LIN {X 0,Y 600.839,Z 923.03,A -85,B 0,C 180,E1 7871.021,E2 7871.021} C_VEL
LIN {X 0,Y 600.811,Z 923.03,A -85,B 0,C 180,E1 7876.847,E2 7876.847} C_VEL
LIN {X 0,Y 600.932,Z 923.03,A -85,B 0,C 180,E1 7882.881,E2 7882.881} C_VEL
LIN {X 0,Y 600.969,Z 923.03,A -85,B 0,C 180,E1 7888.765,E2 7888.765} C_VEL
LIN {X 0,Y 601.067,Z 923.03,A -85,B 0,C 180,E1 7893.096,E2 7893.096} C_VEL
LIN {X 0,Y 601.172,Z 923.03,A -85,B 0,C 180,E1 7898.46,E2 7898.46} C_VEL
LIN {X 0,Y 601.119,Z 923.03,A -85,B 0,C 180,E1 7903.949,E2 7903.949} C_VEL
LIN {X 0,Y 601.484,Z 923.03,A -85,B 0,C 180,E1 7909.873,E2 7909.873} C_VEL
LIN {X 0,Y 601.549,Z 923.323,A -85,B 0,C 180,E1 7914.806,E2 7914.806} C_VEL
LIN {X 0,Y 606.229,Z 948.816,A -85,B 0,C 180,E1 7915.27,E2 7915.27} C_VEL
LIN {X 0,Y 606.178,Z 983.388,A -85,B 0,C 180,E1 7915.848,E2 7915.848} C_VEL
LIN {X 0,Y 605.698,Z 1012.075,A -85,B 0,C 180,E1 7916.874,E2 7916.874} C_VEL
LIN {X 0,Y 605.013,Z 1037.452,A -85,B 0,C 180,E1 7918.391,E2 7918.391} C_VEL
LIN {X 0,Y 604.292,Z 1059.313,A -85,B 0,C 180,E1 7920.36,E2 7920.36} C_VEL
LIN {X 0,Y 603.588,Z 1076.615,A -85,B 0,C 180,E1 7922.692,E2 7922.692} C_VEL
LIN {X 0,Y 602.997,Z 1089.111,A -85,B 0,C 180,E1 7925.394,E2 7925.394} C_VEL
LIN {X 0,Y 602.737,Z 1095.415,A -85,B 0,C 180,E1 7928.184,E2 7928.184} C_VEL
LIN {X 0,Y 602.671,Z 1096.34,A -85,B 0,C 180,E1 7930.11,E2 7930.11} C_VEL
LIN {X 0,Y 602.762,Z 1093.764,A -85,B 0,C 180,E1 7932.471,E2 7932.471} C_VEL
LIN {X 0,Y 602.992,Z 1086.371,A -85,B 0,C 180,E1 7934.97,E2 7934.97} C_VEL
LIN {X 0,Y 603.48,Z 1072.244,A -85,B 0,C 180,E1 7937.641,E2 7937.641} C_VEL
LIN {X 0,Y 604.098,Z 1054.164,A -85,B 0,C 180,E1 7939.855,E2 7939.855} C_VEL
LIN {X 0,Y 604.743,Z 1031.678,A -85,B 0,C 180,E1 7941.725,E2 7941.725} C_VEL
LIN {X 0,Y 605.526,Z 1005.59,A -85,B 0,C 180,E1 7943.163,E2 7943.163} C_VEL
LIN {X 0,Y 605.926,Z 976.016,A -85,B 0,C 180,E1 7944.13,E2 7944.13} C_VEL
LIN {X 0,Y 605.053,Z 940.656,A -85,B 0,C 180,E1 7944.678,E2 7944.678} C_VEL
LIN {X 0,Y 601.353,Z 923.03,A -85,B 0,C 180,E1 7945.032,E2 7945.032} C_VEL
LIN {X 0,Y 600.945,Z 923.03,A -85,B 0,C 180,E1 7951.231,E2 7951.231} C_VEL
LIN {X 0,Y 600.916,Z 923.03,A -85,B 0,C 180,E1 7957.124,E2 7957.124} C_VEL
LIN {X 0,Y 600.782,Z 923.03,A -85,B 0,C 180,E1 7963.15,E2 7963.15} C_VEL
LIN {X 0,Y 600.894,Z 923.03,A -85,B 0,C 180,E1 7969.157,E2 7969.157} C_VEL
LIN {X 0,Y 600.916,Z 923.03,A -85,B 0,C 180,E1 7974.652,E2 7974.652} C_VEL
LIN {X 0,Y 600.987,Z 923.03,A -85,B 0,C 180,E1 7979.798,E2 7979.798} C_VEL
LIN {X 0,Y 601.241,Z 923.03,A -85,B 0,C 180,E1 7984.798,E2 7984.798} C_VEL
LIN {X 0,Y 601.281,Z 923.03,A -85,B 0,C 180,E1 7990.919,E2 7990.919} C_VEL
LIN {X 0,Y 601.286,Z 923.03,A -85,B 0,C 180,E1 7995.433,E2 7995.433} C_VEL
LIN {X 0,Y 601.464,Z 923.03,A -85,B 0,C 180,E1 7999.859,E2 7999.859} C_VEL
LIN {X 0,Y 601.588,Z 923.03,A -85,B 0,C 180,E1 8004.221,E2 8004.221} C_VEL
LIN {X 0,Y 601.735,Z 923.03,A -85,B 0,C 180,E1 8008.548,E2 8008.548} C_VEL
LIN {X 0,Y 601.66,Z 923.03,A -85,B 0,C 180,E1 8012.866,E2 8012.866} C_VEL
LIN {X 0,Y 601.578,Z 923.03,A -85,B 0,C 180,E1 8017.202,E2 8017.202} C_VEL
LIN {X 0,Y 601.437,Z 923.03,A -85,B 0,C 180,E1 8023.055,E2 8023.055} C_VEL
LIN {X 0,Y 601.353,Z 923.03,A -85,B 0,C 180,E1 8027.535,E2 8027.535} C_VEL
LIN {X 0,Y 601.192,Z 923.03,A -85,B 0,C 180,E1 8032.134,E2 8032.134} C_VEL
LIN {X 0,Y 601.149,Z 923.03,A -85,B 0,C 180,E1 8036.885,E2 8036.885} C_VEL
LIN {X 0,Y 601.092,Z 923.03,A -85,B 0,C 180,E1 8041.847,E2 8041.847} C_VEL
LIN {X 0,Y 600.927,Z 923.03,A -85,B 0,C 180,E1 8047.101,E2 8047.101} C_VEL
LIN {X 0,Y 600.986,Z 923.03,A -85,B 0,C 180,E1 8053.181,E2 8053.181} C_VEL
LIN {X 0,Y 600.904,Z 923.03,A -85,B 0,C 180,E1 8059.167,E2 8059.167} C_VEL
LIN {X 0,Y 600.891,Z 923.03,A -85,B 0,C 180,E1 8064.66,E2 8064.66} C_VEL
LIN {X 0,Y 601.13,Z 923.03,A -85,B 0,C 180,E1 8070.645,E2 8070.645} C_VEL
LIN {X 0,Y 601.189,Z 923.03,A -85,B 0,C 180,E1 8071.123,E2 8071.123} C_VEL
LIN {X 0,Y 615.049,Z 964.555,A -85,B 0,C 180,E1 8072.72,E2 8072.72} C_VEL
LIN {X 0,Y 613.064,Z 1002.893,A -85,B 0,C 180,E1 8074.095,E2 8074.095} C_VEL
LIN {X 0,Y 610.732,Z 1039.044,A -85,B 0,C 180,E1 8075.978,E2 8075.978} C_VEL
LIN {X 0,Y 608.192,Z 1072.401,A -85,B 0,C 180,E1 8078.343,E2 8078.343} C_VEL
LIN {X 0,Y 605.791,Z 1103.466,A -85,B 0,C 180,E1 8081.305,E2 8081.305} C_VEL
LIN {X 0,Y 604.138,Z 1128.033,A -85,B 0,C 180,E1 8084.447,E2 8084.447} C_VEL
LIN {X 0,Y 602.911,Z 1147.172,A -85,B 0,C 180,E1 8087.731,E2 8087.731} C_VEL
LIN {X 0,Y 602.274,Z 1162.011,A -85,B 0,C 180,E1 8091.34,E2 8091.34} C_VEL
LIN {X 0,Y 601.991,Z 1171.367,A -85,B 0,C 180,E1 8094.958,E2 8094.958} C_VEL
LIN {X 0,Y 601.888,Z 1175.651,A -85,B 0,C 180,E1 8098.56,E2 8098.56} C_VEL
LIN {X 0,Y 601.892,Z 1175.605,A -85,B 0,C 180,E1 8101.437,E2 8101.437} C_VEL
LIN {X 0,Y 602.053,Z 1171.28,A -85,B 0,C 180,E1 8105.038,E2 8105.038} C_VEL
LIN {X 0,Y 602.289,Z 1161.868,A -85,B 0,C 180,E1 8108.656,E2 8108.656} C_VEL
LIN {X 0,Y 602.951,Z 1146.84,A -85,B 0,C 180,E1 8112.287,E2 8112.287} C_VEL
LIN {X 0,Y 604.213,Z 1126.109,A -85,B 0,C 180,E1 8115.767,E2 8115.767} C_VEL
LIN {X 0,Y 605.984,Z 1100.522,A -85,B 0,C 180,E1 8118.914,E2 8118.914} C_VEL
LIN {X 0,Y 608.17,Z 1070.791,A -85,B 0,C 180,E1 8121.65,E2 8121.65} C_VEL
LIN {X 0,Y 610.558,Z 1037.737,A -85,B 0,C 180,E1 8123.925,E2 8123.925} C_VEL
LIN {X 0,Y 612.697,Z 1001.543,A -85,B 0,C 180,E1 8125.747,E2 8125.747} C_VEL
LIN {X 0,Y 613.951,Z 963.531,A -85,B 0,C 180,E1 8127.081,E2 8127.081} C_VEL
LIN {X 0,Y 601.155,Z 923.03,A -85,B 0,C 180,E1 8128.626,E2 8128.626} C_VEL
LIN {X 0,Y 601.011,Z 923.03,A -85,B 0,C 180,E1 8133.962,E2 8133.962} C_VEL
LIN {X 0,Y 600.872,Z 923.03,A -85,B 0,C 180,E1 8138.953,E2 8138.953} C_VEL
LIN {X 0,Y 600.837,Z 923.03,A -85,B 0,C 180,E1 8140.89,E2 8140.89} C_VEL
LIN {X 0,Y 599.556,Z 923.03,A -85,B 0,C 180,E1 8141.715,E2 8141.715} C_VEL
LIN {X 0,Y 592.929,Z 923.03,A -85,B 0,C 180,E1 8143.956,E2 8143.956} C_VEL
LIN {X 0,Y 592.846,Z 923.03,A -85,B 0,C 180,E1 8144.169,E2 8144.169} C_VEL
LIN {X 0,Y 592.915,Z 923.03,A -85,B 0,C 180,E1 8149.867,E2 8149.867} C_VEL
LIN {X 0,Y 593.127,Z 923.03,A -85,B 0,C 180,E1 8154.61,E2 8154.61} C_VEL
LIN {X 0,Y 593.112,Z 923.03,A -85,B 0,C 180,E1 8160.269,E2 8160.269} C_VEL
LIN {X 0,Y 608.042,Z 967.522,A -85,B 0,C 180,E1 8161.664,E2 8161.664} C_VEL
LIN {X 0,Y 606.659,Z 1011.398,A -85,B 0,C 180,E1 8162.505,E2 8162.505} C_VEL
LIN {X 0,Y 604.629,Z 1052.765,A -85,B 0,C 180,E1 8163.898,E2 8163.898} C_VEL
LIN {X 0,Y 602.308,Z 1090.442,A -85,B 0,C 180,E1 8165.76,E2 8165.76} C_VEL
LIN {X 0,Y 599.934,Z 1125.316,A -85,B 0,C 180,E1 8168.121,E2 8168.121} C_VEL
LIN {X 0,Y 597.69,Z 1156.933,A -85,B 0,C 180,E1 8170.983,E2 8170.983} C_VEL
LIN {X 0,Y 595.986,Z 1183.561,A -85,B 0,C 180,E1 8174.209,E2 8174.209} C_VEL
LIN {X 0,Y 594.902,Z 1204.715,A -85,B 0,C 180,E1 8177.707,E2 8177.707} C_VEL
LIN {X 0,Y 594.348,Z 1219.788,A -85,B 0,C 180,E1 8181.239,E2 8181.239} C_VEL
LIN {X 0,Y 594.132,Z 1229.686,A -85,B 0,C 180,E1 8184.906,E2 8184.906} C_VEL
LIN {X 0,Y 594.006,Z 1234.224,A -85,B 0,C 180,E1 8188.555,E2 8188.555} C_VEL
LIN {X 0,Y 594.127,Z 1234.236,A -85,B 0,C 180,E1 8191.47,E2 8191.47} C_VEL
LIN {X 0,Y 594.141,Z 1229.748,A -85,B 0,C 180,E1 8195.119,E2 8195.119} C_VEL
LIN {X 0,Y 594.374,Z 1219.948,A -85,B 0,C 180,E1 8198.786,E2 8198.786} C_VEL
LIN {X 0,Y 594.984,Z 1204.01,A -85,B 0,C 180,E1 8202.536,E2 8202.536} C_VEL
LIN {X 0,Y 596.173,Z 1183.005,A -85,B 0,C 180,E1 8206.006,E2 8206.006} C_VEL
LIN {X 0,Y 597.992,Z 1157.056,A -85,B 0,C 180,E1 8209.19,E2 8209.19} C_VEL
LIN {X 0,Y 600.341,Z 1126.206,A -85,B 0,C 180,E1 8212.046,E2 8212.046} C_VEL
LIN {X 0,Y 602.999,Z 1091.774,A -85,B 0,C 180,E1 8214.435,E2 8214.435} C_VEL
LIN {X 0,Y 605.496,Z 1055.147,A -85,B 0,C 180,E1 8216.294,E2 8216.294} C_VEL
LIN {X 0,Y 607.732,Z 1015.786,A -85,B 0,C 180,E1 8217.658,E2 8217.658} C_VEL
LIN {X 0,Y 609.171,Z 974.132,A -85,B 0,C 180,E1 8218.5,E2 8218.5} C_VEL
LIN {X 0,Y 608.398,Z 964.807,A -85,B 0,C 180,E1 8218.666,E2 8218.666} C_VEL
LIN {X 0,Y 593.159,Z 923.03,A -85,B 0,C 180,E1 8219.987,E2 8219.987} C_VEL
LIN {X 0,Y 593.061,Z 923.03,A -85,B 0,C 180,E1 8225.888,E2 8225.888} C_VEL
LIN {X 0,Y 592.896,Z 923.03,A -85,B 0,C 180,E1 8231.515,E2 8231.515} C_VEL
LIN {X 0,Y 592.87,Z 923.03,A -85,B 0,C 180,E1 8236.517,E2 8236.517} C_VEL
LIN {X 0,Y 592.972,Z 923.03,A -85,B 0,C 180,E1 8242.297,E2 8242.297} C_VEL
LIN {X 0,Y 593.014,Z 923.03,A -85,B 0,C 180,E1 8247.65,E2 8247.65} C_VEL
LIN {X 0,Y 593.197,Z 923.03,A -85,B 0,C 180,E1 8253.09,E2 8253.09} C_VEL
LIN {X 0,Y 593.241,Z 923.03,A -85,B 0,C 180,E1 8257.539,E2 8257.539} C_VEL
LIN {X 0,Y 593.162,Z 923.03,A -85,B 0,C 180,E1 8262.201,E2 8262.201} C_VEL
LIN {X 0,Y 593.359,Z 923.03,A -85,B 0,C 180,E1 8266.752,E2 8266.752} C_VEL
LIN {X 0,Y 593.633,Z 923.03,A -85,B 0,C 180,E1 8271.216,E2 8271.216} C_VEL
LIN {X 0,Y 593.674,Z 923.03,A -85,B 0,C 180,E1 8274.57,E2 8274.57} C_VEL
LIN {X 0,Y 598.641,Z 949.1,A -85,B 0,C 180,E1 8275.069,E2 8275.069} C_VEL
LIN {X 0,Y 598.556,Z 985.6,A -85,B 0,C 180,E1 8275.704,E2 8275.704} C_VEL
LIN {X 0,Y 597.994,Z 1014.937,A -85,B 0,C 180,E1 8276.799,E2 8276.799} C_VEL
LIN {X 0,Y 597.269,Z 1040.755,A -85,B 0,C 180,E1 8278.416,E2 8278.416} C_VEL
LIN {X 0,Y 596.536,Z 1061.495,A -85,B 0,C 180,E1 8280.364,E2 8280.364} C_VEL
LIN {X 0,Y 595.798,Z 1078.379,A -85,B 0,C 180,E1 8282.727,E2 8282.727} C_VEL
LIN {X 0,Y 595.178,Z 1090.542,A -85,B 0,C 180,E1 8285.465,E2 8285.465} C_VEL
LIN {X 0,Y 594.942,Z 1095.937,A -85,B 0,C 180,E1 8287.823,E2 8287.823} C_VEL
LIN {X 0,Y 594.827,Z 1097.225,A -85,B 0,C 180,E1 8290.245,E2 8290.245} C_VEL
LIN {X 0,Y 594.927,Z 1094.162,A -85,B 0,C 180,E1 8292.718,E2 8292.718} C_VEL
LIN {X 0,Y 595.185,Z 1086.391,A -85,B 0,C 180,E1 8295.225,E2 8295.225} C_VEL
LIN {X 0,Y 595.693,Z 1073.073,A -85,B 0,C 180,E1 8297.724,E2 8297.724} C_VEL
LIN {X 0,Y 596.316,Z 1055.103,A -85,B 0,C 180,E1 8299.948,E2 8299.948} C_VEL
LIN {X 0,Y 597,Z 1032.853,A -85,B 0,C 180,E1 8301.826,E2 8301.826} C_VEL
LIN {X 0,Y 597.811,Z 1006.241,A -85,B 0,C 180,E1 8303.312,E2 8303.312} C_VEL
LIN {X 0,Y 598.239,Z 977.995,A -85,B 0,C 180,E1 8304.258,E2 8304.258} C_VEL
LIN {X 0,Y 597.427,Z 942.053,A -85,B 0,C 180,E1 8304.83,E2 8304.83} C_VEL
LIN {X 0,Y 593.406,Z 923.03,A -85,B 0,C 180,E1 8305.245,E2 8305.245} C_VEL
LIN {X 0,Y 593.037,Z 923.03,A -85,B 0,C 180,E1 8310.64,E2 8310.64} C_VEL
LIN {X 0,Y 593.023,Z 923.03,A -85,B 0,C 180,E1 8315.88,E2 8315.88} C_VEL
LIN {X 0,Y 592.86,Z 923.03,A -85,B 0,C 180,E1 8321.508,E2 8321.508} C_VEL
LIN {X 0,Y 592.881,Z 923.03,A -85,B 0,C 180,E1 8326.503,E2 8326.503} C_VEL
LIN {X 0,Y 592.974,Z 923.03,A -85,B 0,C 180,E1 8332.283,E2 8332.283} C_VEL
LIN {X 0,Y 593,Z 923.03,A -85,B 0,C 180,E1 8337.636,E2 8337.636} C_VEL
LIN {X 0,Y 593.274,Z 923.03,A -85,B 0,C 180,E1 8343.062,E2 8343.062} C_VEL
LIN {X 0,Y 593.316,Z 923.03,A -85,B 0,C 180,E1 8349.099,E2 8349.099} C_VEL
LIN {X 0,Y 593.421,Z 923.03,A -85,B 0,C 180,E1 8353.722,E2 8353.722} C_VEL
LIN {X 0,Y 593.567,Z 923.03,A -85,B 0,C 180,E1 8359.723,E2 8359.723} C_VEL
LIN {X 0,Y 593.68,Z 923.03,A -85,B 0,C 180,E1 8364.144,E2 8364.144} C_VEL
LIN {X 0,Y 593.835,Z 923.03,A -85,B 0,C 180,E1 8368.529,E2 8368.529} C_VEL
LIN {X 0,Y 593.757,Z 923.03,A -85,B 0,C 180,E1 8372.904,E2 8372.904} C_VEL
LIN {X 0,Y 593.69,Z 923.03,A -85,B 0,C 180,E1 8377.298,E2 8377.298} C_VEL
LIN {X 0,Y 593.515,Z 923.03,A -85,B 0,C 180,E1 8383.232,E2 8383.232} C_VEL
LIN {X 0,Y 593.417,Z 923.03,A -85,B 0,C 180,E1 8387.777,E2 8387.777} C_VEL
LIN {X 0,Y 593.266,Z 923.03,A -85,B 0,C 180,E1 8393.512,E2 8393.512} C_VEL
LIN {X 0,Y 593.163,Z 923.03,A -85,B 0,C 180,E1 8398.931,E2 8398.931} C_VEL
LIN {X 0,Y 593.076,Z 923.03,A -85,B 0,C 180,E1 8404.074,E2 8404.074} C_VEL
LIN {X 0,Y 592.976,Z 923.03,A -85,B 0,C 180,E1 8410.135,E2 8410.135} C_VEL
LIN {X 0,Y 593.042,Z 923.03,A -85,B 0,C 180,E1 8415.493,E2 8415.493} C_VEL
LIN {X 0,Y 592.96,Z 923.03,A -85,B 0,C 180,E1 8420.422,E2 8420.422} C_VEL
LIN {X 0,Y 592.984,Z 923.03,A -85,B 0,C 180,E1 8425.899,E2 8425.899} C_VEL
LIN {X 0,Y 593.252,Z 923.03,A -85,B 0,C 180,E1 8430.77,E2 8430.77} C_VEL
LIN {X 0,Y 606.588,Z 962.66,A -85,B 0,C 180,E1 8432.292,E2 8432.292} C_VEL
LIN {X 0,Y 607.639,Z 971.467,A -85,B 0,C 180,E1 8432.613,E2 8432.613} C_VEL
LIN {X 0,Y 605.368,Z 1010.118,A -85,B 0,C 180,E1 8434.12,E2 8434.12} C_VEL
LIN {X 0,Y 602.904,Z 1045.237,A -85,B 0,C 180,E1 8436.081,E2 8436.081} C_VEL
LIN {X 0,Y 600.27,Z 1077.861,A -85,B 0,C 180,E1 8438.542,E2 8438.542} C_VEL
LIN {X 0,Y 597.891,Z 1106.529,A -85,B 0,C 180,E1 8441.413,E2 8441.413} C_VEL
LIN {X 0,Y 596.236,Z 1130.448,A -85,B 0,C 180,E1 8444.595,E2 8444.595} C_VEL
LIN {X 0,Y 595.021,Z 1149.05,A -85,B 0,C 180,E1 8447.921,E2 8447.921} C_VEL
LIN {X 0,Y 594.384,Z 1163.562,A -85,B 0,C 180,E1 8451.63,E2 8451.63} C_VEL
LIN {X 0,Y 594.104,Z 1171.715,A -85,B 0,C 180,E1 8454.891,E2 8454.891} C_VEL
LIN {X 0,Y 593.997,Z 1176.028,A -85,B 0,C 180,E1 8458.541,E2 8458.541} C_VEL
LIN {X 0,Y 594.002,Z 1175.994,A -85,B 0,C 180,E1 8461.456,E2 8461.456} C_VEL
LIN {X 0,Y 594.166,Z 1171.662,A -85,B 0,C 180,E1 8465.105,E2 8465.105} C_VEL
LIN {X 0,Y 594.432,Z 1162.222,A -85,B 0,C 180,E1 8468.772,E2 8468.772} C_VEL
LIN {X 0,Y 595.182,Z 1147.096,A -85,B 0,C 180,E1 8472.45,E2 8472.45} C_VEL
LIN {X 0,Y 596.513,Z 1125.857,A -85,B 0,C 180,E1 8476.029,E2 8476.029} C_VEL
LIN {X 0,Y 598.377,Z 1100.484,A -85,B 0,C 180,E1 8479.164,E2 8479.164} C_VEL
LIN {X 0,Y 600.701,Z 1070.721,A -85,B 0,C 180,E1 8481.922,E2 8481.922} C_VEL
LIN {X 0,Y 603.145,Z 1038.13,A -85,B 0,C 180,E1 8484.186,E2 8484.186} C_VEL
LIN {X 0,Y 605.376,Z 1002.436,A -85,B 0,C 180,E1 8486.008,E2 8486.008} C_VEL
LIN {X 0,Y 606.568,Z 965.188,A -85,B 0,C 180,E1 8487.351,E2 8487.351} C_VEL
LIN {X 0,Y 593.251,Z 923.03,A -85,B 0,C 180,E1 8489.01,E2 8489.01} C_VEL
LIN {X 0,Y 593.096,Z 923.03,A -85,B 0,C 180,E1 8494.09,E2 8494.09} C_VEL
LIN {X 0,Y 592.889,Z 923.03,A -85,B 0,C 180,E1 8500.154,E2 8500.154} C_VEL
LIN {X 0,Y 592.846,Z 923.03,A -85,B 0,C 180,E1 8504.169,E2 8504.169} C_VEL
LIN {X 0,Y 590.332,Z 923.03,A -85,B 0,C 180,E1 8505.418,E2 8505.418} C_VEL
LIN {X 0,Y 585.013,Z 923.03,A -85,B 0,C 180,E1 8507.288,E2 8507.288} C_VEL
LIN {X 0,Y 584.936,Z 923.03,A -85,B 0,C 180,E1 8507.504,E2 8507.504} C_VEL
LIN {X 0,Y 585.103,Z 923.03,A -85,B 0,C 180,E1 8513.579,E2 8513.579} C_VEL
LIN {X 0,Y 585.108,Z 923.03,A -85,B 0,C 180,E1 8518.919,E2 8518.919} C_VEL
LIN {X 0,Y 585.221,Z 923.832,A -85,B 0,C 180,E1 8519.878,E2 8519.878} C_VEL
LIN {X 0,Y 600.717,Z 968.424,A -85,B 0,C 180,E1 8521.349,E2 8521.349} C_VEL
LIN {X 0,Y 599.355,Z 1012.032,A -85,B 0,C 180,E1 8522.228,E2 8522.228} C_VEL
LIN {X 0,Y 597.227,Z 1051.908,A -85,B 0,C 180,E1 8523.592,E2 8523.592} C_VEL
LIN {X 0,Y 594.872,Z 1088.957,A -85,B 0,C 180,E1 8525.437,E2 8525.437} C_VEL
LIN {X 0,Y 592.385,Z 1123.725,A -85,B 0,C 180,E1 8527.799,E2 8527.799} C_VEL
LIN {X 0,Y 590.099,Z 1154.409,A -85,B 0,C 180,E1 8530.571,E2 8530.571} C_VEL
LIN {X 0,Y 588.384,Z 1179.9,A -85,B 0,C 180,E1 8533.605,E2 8533.605} C_VEL
LIN {X 0,Y 587.153,Z 1201.242,A -85,B 0,C 180,E1 8537.001,E2 8537.001} C_VEL
LIN {X 0,Y 586.533,Z 1216.535,A -85,B 0,C 180,E1 8540.374,E2 8540.374} C_VEL
LIN {X 0,Y 586.243,Z 1227.644,A -85,B 0,C 180,E1 8544.096,E2 8544.096} C_VEL
LIN {X 0,Y 586.156,Z 1232.583,A -85,B 0,C 180,E1 8547.058,E2 8547.058} C_VEL
LIN {X 0,Y 586.159,Z 1234.269,A -85,B 0,C 180,E1 8550.013,E2 8550.013} C_VEL
LIN {X 0,Y 586.142,Z 1231.745,A -85,B 0,C 180,E1 8553.708,E2 8553.708} C_VEL
LIN {X 0,Y 586.328,Z 1224.067,A -85,B 0,C 180,E1 8557.416,E2 8557.416} C_VEL
LIN {X 0,Y 586.802,Z 1210.807,A -85,B 0,C 180,E1 8561.148,E2 8561.148} C_VEL
LIN {X 0,Y 587.819,Z 1191.119,A -85,B 0,C 180,E1 8564.908,E2 8564.908} C_VEL
LIN {X 0,Y 589.562,Z 1165.631,A -85,B 0,C 180,E1 8568.406,E2 8568.406} C_VEL
LIN {X 0,Y 591.892,Z 1137.261,A -85,B 0,C 180,E1 8571.328,E2 8571.328} C_VEL
LIN {X 0,Y 594.48,Z 1104.527,A -85,B 0,C 180,E1 8573.883,E2 8573.883} C_VEL
LIN {X 0,Y 597.256,Z 1068.104,A -85,B 0,C 180,E1 8575.985,E2 8575.985} C_VEL
LIN {X 0,Y 599.829,Z 1029.624,A -85,B 0,C 180,E1 8577.542,E2 8577.542} C_VEL
LIN {X 0,Y 601.584,Z 990.606,A -85,B 0,C 180,E1 8578.549,E2 8578.549} C_VEL
LIN {X 0,Y 601.473,Z 967.455,A -85,B 0,C 180,E1 8578.945,E2 8578.945} C_VEL
LIN {X 0,Y 585.234,Z 923.03,A -85,B 0,C 180,E1 8580.427,E2 8580.427} C_VEL
LIN {X 0,Y 585.173,Z 923.03,A -85,B 0,C 180,E1 8584.631,E2 8584.631} C_VEL
LIN {X 0,Y 585.011,Z 923.03,A -85,B 0,C 180,E1 8590.235,E2 8590.235} C_VEL
LIN {X 0,Y 584.963,Z 923.03,A -85,B 0,C 180,E1 8596.341,E2 8596.341} C_VEL
LIN {X 0,Y 585.009,Z 923.03,A -85,B 0,C 180,E1 8601.691,E2 8601.691} C_VEL
LIN {X 0,Y 585.106,Z 923.03,A -85,B 0,C 180,E1 8607.158,E2 8607.158} C_VEL
LIN {X 0,Y 585.178,Z 923.03,A -85,B 0,C 180,E1 8612.304,E2 8612.304} C_VEL
LIN {X 0,Y 585.319,Z 923.03,A -85,B 0,C 180,E1 8617.218,E2 8617.218} C_VEL
LIN {X 0,Y 585.267,Z 923.03,A -85,B 0,C 180,E1 8622.831,E2 8622.831} C_VEL
LIN {X 0,Y 585.575,Z 923.03,A -85,B 0,C 180,E1 8628.736,E2 8628.736} C_VEL
LIN {X 0,Y 585.764,Z 923.03,A -85,B 0,C 180,E1 8634.311,E2 8634.311} C_VEL
LIN {X 0,Y 591.065,Z 950.012,A -85,B 0,C 180,E1 8634.868,E2 8634.868} C_VEL
LIN {X 0,Y 590.958,Z 986.526,A -85,B 0,C 180,E1 8635.51,E2 8635.51} C_VEL
LIN {X 0,Y 590.378,Z 1015.616,A -85,B 0,C 180,E1 8636.608,E2 8636.608} C_VEL
LIN {X 0,Y 589.616,Z 1041.655,A -85,B 0,C 180,E1 8638.258,E2 8638.258} C_VEL
LIN {X 0,Y 588.859,Z 1062.054,A -85,B 0,C 180,E1 8640.185,E2 8640.185} C_VEL
LIN {X 0,Y 588.043,Z 1079.108,A -85,B 0,C 180,E1 8642.579,E2 8642.579} C_VEL
LIN {X 0,Y 587.414,Z 1090.749,A -85,B 0,C 180,E1 8645.167,E2 8645.167} C_VEL
LIN {X 0,Y 587.143,Z 1096.322,A -85,B 0,C 180,E1 8647.395,E2 8647.395} C_VEL
LIN {X 0,Y 586.992,Z 1098.11,A -85,B 0,C 180,E1 8650.383,E2 8650.383} C_VEL
LIN {X 0,Y 587.1,Z 1094.473,A -85,B 0,C 180,E1 8652.979,E2 8652.979} C_VEL
LIN {X 0,Y 587.437,Z 1085.55,A -85,B 0,C 180,E1 8655.682,E2 8655.682} C_VEL
LIN {X 0,Y 588.003,Z 1070.16,A -85,B 0,C 180,E1 8658.35,E2 8658.35} C_VEL
LIN {X 0,Y 588.748,Z 1051.052,A -85,B 0,C 180,E1 8660.532,E2 8660.532} C_VEL
LIN {X 0,Y 589.522,Z 1026.602,A -85,B 0,C 180,E1 8662.415,E2 8662.415} C_VEL
LIN {X 0,Y 590.225,Z 998.779,A -85,B 0,C 180,E1 8663.797,E2 8663.797} C_VEL
LIN {X 0,Y 590.596,Z 967.955,A -85,B 0,C 180,E1 8664.628,E2 8664.628} C_VEL
LIN {X 0,Y 589.648,Z 942.756,A -85,B 0,C 180,E1 8664.996,E2 8664.996} C_VEL
LIN {X 0,Y 585.47,Z 923.03,A -85,B 0,C 180,E1 8665.379,E2 8665.379} C_VEL
LIN {X 0,Y 585.053,Z 923.03,A -85,B 0,C 180,E1 8671.517,E2 8671.517} C_VEL
LIN {X 0,Y 585.033,Z 923.03,A -85,B 0,C 180,E1 8676.788,E2 8676.788} C_VEL
LIN {X 0,Y 584.943,Z 923.03,A -85,B 0,C 180,E1 8682.198,E2 8682.198} C_VEL
LIN {X 0,Y 584.998,Z 923.03,A -85,B 0,C 180,E1 8687.797,E2 8687.797} C_VEL
LIN {X 0,Y 585.039,Z 923.03,A -85,B 0,C 180,E1 8693.542,E2 8693.542} C_VEL
LIN {X 0,Y 585.103,Z 923.03,A -85,B 0,C 180,E1 8698.889,E2 8698.889} C_VEL
LIN {X 0,Y 585.331,Z 923.03,A -85,B 0,C 180,E1 8704.634,E2 8704.634} C_VEL
LIN {X 0,Y 585.43,Z 923.03,A -85,B 0,C 180,E1 8710.382,E2 8710.382} C_VEL
LIN {X 0,Y 585.46,Z 923.03,A -85,B 0,C 180,E1 8715.03,E2 8715.03} C_VEL
LIN {X 0,Y 585.643,Z 923.03,A -85,B 0,C 180,E1 8719.582,E2 8719.582} C_VEL
LIN {X 0,Y 585.806,Z 923.03,A -85,B 0,C 180,E1 8724.065,E2 8724.065} C_VEL
LIN {X 0,Y 585.934,Z 923.03,A -85,B 0,C 180,E1 8728.509,E2 8728.509} C_VEL
LIN {X 0,Y 585.856,Z 923.03,A -85,B 0,C 180,E1 8732.944,E2 8732.944} C_VEL
LIN {X 0,Y 585.776,Z 923.03,A -85,B 0,C 180,E1 8737.397,E2 8737.397} C_VEL
LIN {X 0,Y 585.608,Z 923.03,A -85,B 0,C 180,E1 8743.414,E2 8743.414} C_VEL
LIN {X 0,Y 585.502,Z 923.03,A -85,B 0,C 180,E1 8748.026,E2 8748.026} C_VEL
LIN {X 0,Y 585.335,Z 923.03,A -85,B 0,C 180,E1 8752.766,E2 8752.766} C_VEL
LIN {X 0,Y 585.264,Z 923.03,A -85,B 0,C 180,E1 8758.613,E2 8758.613} C_VEL
LIN {X 0,Y 585.164,Z 923.03,A -85,B 0,C 180,E1 8764.599,E2 8764.599} C_VEL
LIN {X 0,Y 585.076,Z 923.03,A -85,B 0,C 180,E1 8770.195,E2 8770.195} C_VEL
LIN {X 0,Y 585.132,Z 923.03,A -85,B 0,C 180,E1 8775.789,E2 8775.789} C_VEL
LIN {X 0,Y 585.002,Z 923.03,A -85,B 0,C 180,E1 8781.687,E2 8781.687} C_VEL
LIN {X 0,Y 585.079,Z 923.03,A -85,B 0,C 180,E1 8787.153,E2 8787.153} C_VEL
LIN {X 0,Y 585.351,Z 923.785,A -85,B 0,C 180,E1 8790.407,E2 8790.407} C_VEL
LIN {X 0,Y 598.951,Z 963.422,A -85,B 0,C 180,E1 8791.971,E2 8791.971} C_VEL
LIN {X 0,Y 600.452,Z 971.844,A -85,B 0,C 180,E1 8792.307,E2 8792.307} C_VEL
LIN {X 0,Y 598.023,Z 1010.969,A -85,B 0,C 180,E1 8793.856,E2 8793.856} C_VEL
LIN {X 0,Y 595.384,Z 1046.785,A -85,B 0,C 180,E1 8795.894,E2 8795.894} C_VEL
LIN {X 0,Y 592.716,Z 1078.64,A -85,B 0,C 180,E1 8798.34,E2 8798.34} C_VEL
LIN {X 0,Y 590.187,Z 1107.402,A -85,B 0,C 180,E1 8801.266,E2 8801.266} C_VEL
LIN {X 0,Y 588.497,Z 1130.788,A -85,B 0,C 180,E1 8804.423,E2 8804.423} C_VEL
LIN {X 0,Y 587.176,Z 1149.703,A -85,B 0,C 180,E1 8807.853,E2 8807.853} C_VEL
LIN {X 0,Y 586.52,Z 1163.737,A -85,B 0,C 180,E1 8811.479,E2 8811.479} C_VEL
LIN {X 0,Y 586.219,Z 1172.062,A -85,B 0,C 180,E1 8814.822,E2 8814.822} C_VEL
LIN {X 0,Y 586.127,Z 1176.404,A -85,B 0,C 180,E1 8818.521,E2 8818.521} C_VEL
LIN {X 0,Y 586.132,Z 1176.382,A -85,B 0,C 180,E1 8821.476,E2 8821.476} C_VEL
LIN {X 0,Y 586.295,Z 1172.039,A -85,B 0,C 180,E1 8825.174,E2 8825.174} C_VEL
LIN {X 0,Y 586.587,Z 1162.566,A -85,B 0,C 180,E1 8828.89,E2 8828.89} C_VEL
LIN {X 0,Y 587.409,Z 1146.94,A -85,B 0,C 180,E1 8832.695,E2 8832.695} C_VEL
LIN {X 0,Y 588.832,Z 1125.985,A -85,B 0,C 180,E1 8836.244,E2 8836.244} C_VEL
LIN {X 0,Y 590.779,Z 1100.486,A -85,B 0,C 180,E1 8839.42,E2 8839.42} C_VEL
LIN {X 0,Y 593.185,Z 1071.329,A -85,B 0,C 180,E1 8842.151,E2 8842.151} C_VEL
LIN {X 0,Y 595.732,Z 1038.857,A -85,B 0,C 180,E1 8844.44,E2 8844.44} C_VEL
LIN {X 0,Y 598.151,Z 1002.052,A -85,B 0,C 180,E1 8846.338,E2 8846.338} C_VEL
LIN {X 0,Y 599.29,Z 967.203,A -85,B 0,C 180,E1 8847.619,E2 8847.619} C_VEL
LIN {X 0,Y 586.769,Z 927.616,A -85,B 0,C 180,E1 8849.206,E2 8849.206} C_VEL
LIN {X 0,Y 585.356,Z 923.03,A -85,B 0,C 180,E1 8849.371,E2 8849.371} C_VEL
LIN {X 0,Y 585.171,Z 923.03,A -85,B 0,C 180,E1 8854.617,E2 8854.617} C_VEL
LIN {X 0,Y 584.987,Z 923.03,A -85,B 0,C 180,E1 8860.222,E2 8860.222} C_VEL
LIN {X 0,Y 584.965,Z 923.03,A -85,B 0,C 180,E1 8866.326,E2 8866.326} C_VEL
LIN {X 0,Y 584.936,Z 923.03,A -85,B 0,C 180,E1 8867.504,E2 8867.504} C_VEL
LIN {X 0,Y 582.445,Z 923.03,A -85,B 0,C 180,E1 8868.768,E2 8868.768} C_VEL
LIN {X 0,Y 577.15,Z 923.03,A -85,B 0,C 180,E1 8870.66,E2 8870.66} C_VEL
LIN {X 0,Y 577.081,Z 923.03,A -85,B 0,C 180,E1 8870.879,E2 8870.879} C_VEL
LIN {X 0,Y 577.206,Z 923.03,A -85,B 0,C 180,E1 8876.9,E2 8876.9} C_VEL
LIN {X 0,Y 577.239,Z 923.115,A -85,B 0,C 180,E1 8879.405,E2 8879.405} C_VEL
LIN {X 0,Y 591.158,Z 963.17,A -85,B 0,C 180,E1 8880.816,E2 8880.816} C_VEL
LIN {X 0,Y 593.655,Z 973.013,A -85,B 0,C 180,E1 8881.095,E2 8881.095} C_VEL
LIN {X 0,Y 591.963,Z 1015.439,A -85,B 0,C 180,E1 8882.019,E2 8882.019} C_VEL
LIN {X 0,Y 589.617,Z 1056.219,A -85,B 0,C 180,E1 8883.499,E2 8883.499} C_VEL
LIN {X 0,Y 586.973,Z 1094.02,A -85,B 0,C 180,E1 8885.49,E2 8885.49} C_VEL
LIN {X 0,Y 584.262,Z 1129.871,A -85,B 0,C 180,E1 8888.091,E2 8888.091} C_VEL
LIN {X 0,Y 581.948,Z 1159.976,A -85,B 0,C 180,E1 8891.012,E2 8891.012} C_VEL
LIN {X 0,Y 580.241,Z 1184.592,A -85,B 0,C 180,E1 8894.165,E2 8894.165} C_VEL
LIN {X 0,Y 579.127,Z 1204.486,A -85,B 0,C 180,E1 8897.584,E2 8897.584} C_VEL
LIN {X 0,Y 578.557,Z 1219.966,A -85,B 0,C 180,E1 8901.377,E2 8901.377} C_VEL
LIN {X 0,Y 578.373,Z 1228.808,A -85,B 0,C 180,E1 8904.767,E2 8904.767} C_VEL
LIN {X 0,Y 578.234,Z 1233.434,A -85,B 0,C 180,E1 8908.516,E2 8908.516} C_VEL
LIN {X 0,Y 578.363,Z 1233.468,A -85,B 0,C 180,E1 8911.51,E2 8911.51} C_VEL
LIN {X 0,Y 578.385,Z 1228.955,A -85,B 0,C 180,E1 8915.259,E2 8915.259} C_VEL
LIN {X 0,Y 578.588,Z 1219.087,A -85,B 0,C 180,E1 8919.028,E2 8919.028} C_VEL
LIN {X 0,Y 579.27,Z 1203.307,A -85,B 0,C 180,E1 8922.823,E2 8922.823} C_VEL
LIN {X 0,Y 580.6,Z 1181.638,A -85,B 0,C 180,E1 8926.474,E2 8926.474} C_VEL
LIN {X 0,Y 582.659,Z 1155.66,A -85,B 0,C 180,E1 8929.715,E2 8929.715} C_VEL
LIN {X 0,Y 585.196,Z 1125.29,A -85,B 0,C 180,E1 8932.58,E2 8932.58} C_VEL
LIN {X 0,Y 588.177,Z 1091.223,A -85,B 0,C 180,E1 8934.992,E2 8934.992} C_VEL
LIN {X 0,Y 590.834,Z 1054.975,A -85,B 0,C 180,E1 8936.877,E2 8936.877} C_VEL
LIN {X 0,Y 593.281,Z 1015.939,A -85,B 0,C 180,E1 8938.268,E2 8938.268} C_VEL
LIN {X 0,Y 594.89,Z 975.29,A -85,B 0,C 180,E1 8939.125,E2 8939.125} C_VEL
LIN {X 0,Y 593.464,Z 966.935,A -85,B 0,C 180,E1 8939.318,E2 8939.318} C_VEL
LIN {X 0,Y 577.321,Z 923.03,A -85,B 0,C 180,E1 8940.82,E2 8940.82} C_VEL
LIN {X 0,Y 577.148,Z 923.03,A -85,B 0,C 180,E1 8945.746,E2 8945.746} C_VEL
LIN {X 0,Y 577.093,Z 923.03,A -85,B 0,C 180,E1 8950.903,E2 8950.903} C_VEL
LIN {X 0,Y 577.024,Z 923.03,A -85,B 0,C 180,E1 8957.174,E2 8957.174} C_VEL
LIN {X 0,Y 577.127,Z 923.03,A -85,B 0,C 180,E1 8962.974,E2 8962.974} C_VEL
LIN {X 0,Y 577.174,Z 923.03,A -85,B 0,C 180,E1 8968.427,E2 8968.427} C_VEL
LIN {X 0,Y 577.289,Z 923.03,A -85,B 0,C 180,E1 8973.579,E2 8973.579} C_VEL
LIN {X 0,Y 577.42,Z 923.03,A -85,B 0,C 180,E1 8978.509,E2 8978.509} C_VEL
LIN {X 0,Y 577.418,Z 923.03,A -85,B 0,C 180,E1 8984.831,E2 8984.831} C_VEL
LIN {X 0,Y 577.749,Z 923.03,A -85,B 0,C 180,E1 8989.452,E2 8989.452} C_VEL
LIN {X 0,Y 577.849,Z 923.592,A -85,B 0,C 180,E1 8994.091,E2 8994.091} C_VEL
LIN {X 0,Y 583.507,Z 951.064,A -85,B 0,C 180,E1 8994.662,E2 8994.662} C_VEL
LIN {X 0,Y 583.383,Z 987.488,A -85,B 0,C 180,E1 8995.312,E2 8995.312} C_VEL
LIN {X 0,Y 582.811,Z 1015.717,A -85,B 0,C 180,E1 8996.378,E2 8996.378} C_VEL
LIN {X 0,Y 582.038,Z 1040.883,A -85,B 0,C 180,E1 8997.956,E2 8997.956} C_VEL
LIN {X 0,Y 581.158,Z 1062.638,A -85,B 0,C 180,E1 9000.002,E2 9000.002} C_VEL
LIN {X 0,Y 580.31,Z 1079.831,A -85,B 0,C 180,E1 9002.427,E2 9002.427} C_VEL
LIN {X 0,Y 579.602,Z 1092.22,A -85,B 0,C 180,E1 9005.237,E2 9005.237} C_VEL
LIN {X 0,Y 579.297,Z 1097.563,A -85,B 0,C 180,E1 9007.534,E2 9007.534} C_VEL
LIN {X 0,Y 579.145,Z 1098.994,A -85,B 0,C 180,E1 9010.525,E2 9010.525} C_VEL
LIN {X 0,Y 579.253,Z 1095.832,A -85,B 0,C 180,E1 9012.813,E2 9012.813} C_VEL
LIN {X 0,Y 579.585,Z 1087.545,A -85,B 0,C 180,E1 9015.463,E2 9015.463} C_VEL
LIN {X 0,Y 580.106,Z 1073.933,A -85,B 0,C 180,E1 9018.008,E2 9018.008} C_VEL
LIN {X 0,Y 580.832,Z 1055.549,A -85,B 0,C 180,E1 9020.276,E2 9020.276} C_VEL
LIN {X 0,Y 581.553,Z 1032.459,A -85,B 0,C 180,E1 9022.212,E2 9022.212} C_VEL
LIN {X 0,Y 582.422,Z 1005.149,A -85,B 0,C 180,E1 9023.714,E2 9023.714} C_VEL
LIN {X 0,Y 582.853,Z 974.925,A -85,B 0,C 180,E1 9024.667,E2 9024.667} C_VEL
LIN {X 0,Y 582.12,Z 944.598,A -85,B 0,C 180,E1 9025.142,E2 9025.142} C_VEL
LIN {X 0,Y 577.521,Z 923.03,A -85,B 0,C 180,E1 9025.586,E2 9025.586} C_VEL
LIN {X 0,Y 577.151,Z 923.03,A -85,B 0,C 180,E1 9031.579,E2 9031.579} C_VEL
LIN {X 0,Y 577.113,Z 923.03,A -85,B 0,C 180,E1 9037.031,E2 9037.031} C_VEL
LIN {X 0,Y 577.015,Z 923.03,A -85,B 0,C 180,E1 9042.916,E2 9042.916} C_VEL
LIN {X 0,Y 577.145,Z 923.03,A -85,B 0,C 180,E1 9049.404,E2 9049.404} C_VEL
LIN {X 0,Y 577.109,Z 923.03,A -85,B 0,C 180,E1 9054.815,E2 9054.815} C_VEL
LIN {X 0,Y 577.209,Z 923.03,A -85,B 0,C 180,E1 9060.159,E2 9060.159} C_VEL
LIN {X 0,Y 577.412,Z 923.03,A -85,B 0,C 180,E1 9065.234,E2 9065.234} C_VEL
LIN {X 0,Y 577.53,Z 923.03,A -85,B 0,C 180,E1 9070.383,E2 9070.383} C_VEL
LIN {X 0,Y 577.534,Z 923.03,A -85,B 0,C 180,E1 9075.493,E2 9075.493} C_VEL
LIN {X 0,Y 577.781,Z 923.03,A -85,B 0,C 180,E1 9080.959,E2 9080.959} C_VEL
LIN {X 0,Y 578.113,Z 923.03,A -85,B 0,C 180,E1 9086.99,E2 9086.99} C_VEL
LIN {X 0,Y 578.121,Z 923.03,A -85,B 0,C 180,E1 9091.484,E2 9091.484} C_VEL
LIN {X 0,Y 577.891,Z 923.03,A -85,B 0,C 180,E1 9097.498,E2 9097.498} C_VEL
LIN {X 0,Y 577.681,Z 923.03,A -85,B 0,C 180,E1 9103.602,E2 9103.602} C_VEL
LIN {X 0,Y 577.562,Z 923.03,A -85,B 0,C 180,E1 9108.282,E2 9108.282} C_VEL
LIN {X 0,Y 577.355,Z 923.03,A -85,B 0,C 180,E1 9113.641,E2 9113.641} C_VEL
LIN {X 0,Y 577.343,Z 923.03,A -85,B 0,C 180,E1 9118.089,E2 9118.089} C_VEL
LIN {X 0,Y 577.242,Z 923.03,A -85,B 0,C 180,E1 9123.33,E2 9123.33} C_VEL
LIN {X 0,Y 577.128,Z 923.03,A -85,B 0,C 180,E1 9128.91,E2 9128.91} C_VEL
LIN {X 0,Y 577.186,Z 923.03,A -85,B 0,C 180,E1 9135.017,E2 9135.017} C_VEL
LIN {X 0,Y 577.114,Z 923.03,A -85,B 0,C 180,E1 9141.065,E2 9141.065} C_VEL
LIN {X 0,Y 577.168,Z 923.03,A -85,B 0,C 180,E1 9146.876,E2 9146.876} C_VEL
LIN {X 0,Y 577.377,Z 923.03,A -85,B 0,C 180,E1 9149.999,E2 9149.999} C_VEL
LIN {X 0,Y 591.308,Z 964.136,A -85,B 0,C 180,E1 9151.649,E2 9151.649} C_VEL
LIN {X 0,Y 593.177,Z 973.53,A -85,B 0,C 180,E1 9152.043,E2 9152.043} C_VEL
LIN {X 0,Y 590.706,Z 1011.801,A -85,B 0,C 180,E1 9153.587,E2 9153.587} C_VEL
LIN {X 0,Y 588.006,Z 1047.053,A -85,B 0,C 180,E1 9155.618,E2 9155.618} C_VEL
LIN {X 0,Y 585.169,Z 1079.35,A -85,B 0,C 180,E1 9158.13,E2 9158.13} C_VEL
LIN {X 0,Y 582.616,Z 1107.387,A -85,B 0,C 180,E1 9161.014,E2 9161.014} C_VEL
LIN {X 0,Y 580.759,Z 1131.07,A -85,B 0,C 180,E1 9164.238,E2 9164.238} C_VEL
LIN {X 0,Y 579.371,Z 1149.915,A -85,B 0,C 180,E1 9167.687,E2 9167.687} C_VEL
LIN {X 0,Y 578.653,Z 1164.029,A -85,B 0,C 180,E1 9171.362,E2 9171.362} C_VEL
LIN {X 0,Y 578.34,Z 1172.407,A -85,B 0,C 180,E1 9174.751,E2 9174.751} C_VEL
LIN {X 0,Y 578.234,Z 1176.781,A -85,B 0,C 180,E1 9178.501,E2 9178.501} C_VEL
LIN {X 0,Y 578.241,Z 1176.772,A -85,B 0,C 180,E1 9181.496,E2 9181.496} C_VEL
LIN {X 0,Y 578.412,Z 1172.415,A -85,B 0,C 180,E1 9185.245,E2 9185.245} C_VEL
LIN {X 0,Y 578.732,Z 1162.902,A -85,B 0,C 180,E1 9189.012,E2 9189.012} C_VEL
LIN {X 0,Y 579.588,Z 1147.535,A -85,B 0,C 180,E1 9192.802,E2 9192.802} C_VEL
LIN {X 0,Y 581.089,Z 1126.853,A -85,B 0,C 180,E1 9196.363,E2 9196.363} C_VEL
LIN {X 0,Y 583.046,Z 1102.363,A -85,B 0,C 180,E1 9199.485,E2 9199.485} C_VEL
LIN {X 0,Y 585.624,Z 1072.579,A -85,B 0,C 180,E1 9202.339,E2 9202.339} C_VEL
LIN {X 0,Y 588.31,Z 1040.171,A -85,B 0,C 180,E1 9204.668,E2 9204.668} C_VEL
LIN {X 0,Y 590.832,Z 1004.146,A -85,B 0,C 180,E1 9206.57,E2 9206.57} C_VEL
LIN {X 0,Y 591.924,Z 968.743,A -85,B 0,C 180,E1 9207.921,E2 9207.921} C_VEL
LIN {X 0,Y 580.067,Z 930.745,A -85,B 0,C 180,E1 9209.516,E2 9209.516} C_VEL
LIN {X 0,Y 577.372,Z 923.03,A -85,B 0,C 180,E1 9209.818,E2 9209.818} C_VEL
LIN {X 0,Y 577.173,Z 923.03,A -85,B 0,C 180,E1 9215.166,E2 9215.166} C_VEL
LIN {X 0,Y 577.07,Z 923.03,A -85,B 0,C 180,E1 9220.89,E2 9220.89} C_VEL
LIN {X 0,Y 577.044,Z 923.03,A -85,B 0,C 180,E1 9227.156,E2 9227.156} C_VEL
LIN {X 0,Y 577.081,Z 923.03,A -85,B 0,C 180,E1 9230.879,E2 9230.879} C_VEL
LIN {X 0,Y 574.699,Z 923.03,A -85,B 0,C 180,E1 9232.16,E2 9232.16} C_VEL
LIN {X 0,Y 569.275,Z 923.03,A -85,B 0,C 180,E1 9234.3,E2 9234.3} C_VEL
LIN {X 0,Y 569.364,Z 923.751,A -85,B 0,C 180,E1 9238.931,E2 9238.931} C_VEL
LIN {X 0,Y 582.625,Z 959.751,A -85,B 0,C 180,E1 9240.324,E2 9240.324} C_VEL
LIN {X 0,Y 586.551,Z 974.88,A -85,B 0,C 180,E1 9240.781,E2 9240.781} C_VEL
LIN {X 0,Y 584.658,Z 1017.2,A -85,B 0,C 180,E1 9241.75,E2 9241.75} C_VEL
LIN {X 0,Y 582.056,Z 1059.278,A -85,B 0,C 180,E1 9243.346,E2 9243.346} C_VEL
LIN {X 0,Y 579.17,Z 1097.456,A -85,B 0,C 180,E1 9245.459,E2 9245.459} C_VEL
LIN {X 0,Y 576.535,Z 1131.044,A -85,B 0,C 180,E1 9247.984,E2 9247.984} C_VEL
LIN {X 0,Y 574.208,Z 1159.471,A -85,B 0,C 180,E1 9250.792,E2 9250.792} C_VEL
LIN {X 0,Y 572.401,Z 1184.261,A -85,B 0,C 180,E1 9254.007,E2 9254.007} C_VEL
LIN {X 0,Y 571.291,Z 1203.864,A -85,B 0,C 180,E1 9257.411,E2 9257.411} C_VEL
LIN {X 0,Y 570.662,Z 1219.45,A -85,B 0,C 180,E1 9261.257,E2 9261.257} C_VEL
LIN {X 0,Y 570.475,Z 1228.366,A -85,B 0,C 180,E1 9264.694,E2 9264.694} C_VEL
LIN {X 0,Y 570.341,Z 1233.038,A -85,B 0,C 180,E1 9268.495,E2 9268.495} C_VEL
LIN {X 0,Y 570.466,Z 1233.083,A -85,B 0,C 180,E1 9271.531,E2 9271.531} C_VEL
LIN {X 0,Y 570.489,Z 1228.557,A -85,B 0,C 180,E1 9275.332,E2 9275.332} C_VEL
LIN {X 0,Y 570.705,Z 1218.654,A -85,B 0,C 180,E1 9279.154,E2 9279.154} C_VEL
LIN {X 0,Y 571.43,Z 1202.801,A -85,B 0,C 180,E1 9283.002,E2 9283.002} C_VEL
LIN {X 0,Y 572.789,Z 1181.806,A -85,B 0,C 180,E1 9286.593,E2 9286.593} C_VEL
LIN {X 0,Y 574.837,Z 1156.831,A -85,B 0,C 180,E1 9289.782,E2 9289.782} C_VEL
LIN {X 0,Y 577.497,Z 1126.515,A -85,B 0,C 180,E1 9292.715,E2 9292.715} C_VEL
LIN {X 0,Y 580.529,Z 1093.175,A -85,B 0,C 180,E1 9295.138,E2 9295.138} C_VEL
LIN {X 0,Y 583.453,Z 1055.728,A -85,B 0,C 180,E1 9297.136,E2 9297.136} C_VEL
LIN {X 0,Y 586.057,Z 1016.292,A -85,B 0,C 180,E1 9298.571,E2 9298.571} C_VEL
LIN {X 0,Y 587.75,Z 976.077,A -85,B 0,C 180,E1 9299.442,E2 9299.442} C_VEL
LIN {X 0,Y 585.387,Z 966.066,A -85,B 0,C 180,E1 9299.71,E2 9299.71} C_VEL
LIN {X 0,Y 569.382,Z 923.03,A -85,B 0,C 180,E1 9301.208,E2 9301.208} C_VEL
LIN {X 0,Y 569.211,Z 923.03,A -85,B 0,C 180,E1 9307.213,E2 9307.213} C_VEL
LIN {X 0,Y 569.078,Z 923.03,A -85,B 0,C 180,E1 9311.972,E2 9311.972} C_VEL
LIN {X 0,Y 569.078,Z 923.03,A -85,B 0,C 180,E1 9318.044,E2 9318.044} C_VEL
LIN {X 0,Y 569.256,Z 923.03,A -85,B 0,C 180,E1 9324.27,E2 9324.27} C_VEL
LIN {X 0,Y 569.266,Z 923.03,A -85,B 0,C 180,E1 9329.714,E2 9329.714} C_VEL
LIN {X 0,Y 569.392,Z 923.03,A -85,B 0,C 180,E1 9334.875,E2 9334.875} C_VEL
LIN {X 0,Y 569.443,Z 923.03,A -85,B 0,C 180,E1 9339.822,E2 9339.822} C_VEL
LIN {X 0,Y 569.487,Z 923.03,A -85,B 0,C 180,E1 9344.614,E2 9344.614} C_VEL
LIN {X 0,Y 569.819,Z 923.03,A -85,B 0,C 180,E1 9349.304,E2 9349.304} C_VEL
LIN {X 0,Y 569.932,Z 923.03,A -85,B 0,C 180,E1 9353.792,E2 9353.792} C_VEL
LIN {X 0,Y 575.951,Z 952.526,A -85,B 0,C 180,E1 9354.45,E2 9354.45} C_VEL
LIN {X 0,Y 575.816,Z 988.483,A -85,B 0,C 180,E1 9355.109,E2 9355.109} C_VEL
LIN {X 0,Y 575.21,Z 1017.599,A -85,B 0,C 180,E1 9356.236,E2 9356.236} C_VEL
LIN {X 0,Y 574.33,Z 1043.711,A -85,B 0,C 180,E1 9357.928,E2 9357.928} C_VEL
LIN {X 0,Y 573.404,Z 1064.885,A -85,B 0,C 180,E1 9360.002,E2 9360.002} C_VEL
LIN {X 0,Y 572.52,Z 1081.65,A -85,B 0,C 180,E1 9362.46,E2 9362.46} C_VEL
LIN {X 0,Y 571.781,Z 1093.654,A -85,B 0,C 180,E1 9365.309,E2 9365.309} C_VEL
LIN {X 0,Y 571.46,Z 1098.692,A -85,B 0,C 180,E1 9367.599,E2 9367.599} C_VEL
LIN {X 0,Y 571.326,Z 1100.07,A -85,B 0,C 180,E1 9369.133,E2 9369.133} C_VEL
LIN {X 0,Y 571.367,Z 1098.57,A -85,B 0,C 180,E1 9371.852,E2 9371.852} C_VEL
LIN {X 0,Y 571.68,Z 1090.698,A -85,B 0,C 180,E1 9374.93,E2 9374.93} C_VEL
LIN {X 0,Y 572.123,Z 1078.568,A -85,B 0,C 180,E1 9377.481,E2 9377.481} C_VEL
LIN {X 0,Y 572.8,Z 1061.251,A -85,B 0,C 180,E1 9379.858,E2 9379.858} C_VEL
LIN {X 0,Y 573.683,Z 1038.529,A -85,B 0,C 180,E1 9381.957,E2 9381.957} C_VEL
LIN {X 0,Y 574.578,Z 1012.799,A -85,B 0,C 180,E1 9383.544,E2 9383.544} C_VEL
LIN {X 0,Y 575.083,Z 984.748,A -85,B 0,C 180,E1 9384.604,E2 9384.604} C_VEL
LIN {X 0,Y 574.516,Z 946.112,A -85,B 0,C 180,E1 9385.295,E2 9385.295} C_VEL
LIN {X 0,Y 569.585,Z 923.03,A -85,B 0,C 180,E1 9385.783,E2 9385.783} C_VEL
LIN {X 0,Y 569.214,Z 923.03,A -85,B 0,C 180,E1 9392.071,E2 9392.071} C_VEL
LIN {X 0,Y 569.183,Z 923.03,A -85,B 0,C 180,E1 9397.636,E2 9397.636} C_VEL
LIN {X 0,Y 569.02,Z 923.03,A -85,B 0,C 180,E1 9403.669,E2 9403.669} C_VEL
LIN {X 0,Y 569.128,Z 923.03,A -85,B 0,C 180,E1 9408.398,E2 9408.398} C_VEL
LIN {X 0,Y 569.221,Z 923.03,A -85,B 0,C 180,E1 9414.253,E2 9414.253} C_VEL
LIN {X 0,Y 569.28,Z 923.03,A -85,B 0,C 180,E1 9419.7,E2 9419.7} C_VEL
LIN {X 0,Y 569.465,Z 923.03,A -85,B 0,C 180,E1 9424.865,E2 9424.865} C_VEL
LIN {X 0,Y 569.56,Z 923.03,A -85,B 0,C 180,E1 9429.812,E2 9429.812} C_VEL
LIN {X 0,Y 569.63,Z 923.03,A -85,B 0,C 180,E1 9434.604,E2 9434.604} C_VEL
LIN {X 0,Y 569.806,Z 923.03,A -85,B 0,C 180,E1 9439.289,E2 9439.289} C_VEL
LIN {X 0,Y 570,Z 923.03,A -85,B 0,C 180,E1 9443.9,E2 9443.9} C_VEL
LIN {X 0,Y 570.137,Z 923.03,A -85,B 0,C 180,E1 9448.468,E2 9448.468} C_VEL
LIN {X 0,Y 570.059,Z 923.03,A -85,B 0,C 180,E1 9453.025,E2 9453.025} C_VEL
LIN {X 0,Y 569.974,Z 923.03,A -85,B 0,C 180,E1 9457.603,E2 9457.603} C_VEL
LIN {X 0,Y 569.765,Z 923.03,A -85,B 0,C 180,E1 9463.794,E2 9463.794} C_VEL
LIN {X 0,Y 569.635,Z 923.03,A -85,B 0,C 180,E1 9468.546,E2 9468.546} C_VEL
LIN {X 0,Y 569.462,Z 923.03,A -85,B 0,C 180,E1 9473.438,E2 9473.438} C_VEL
LIN {X 0,Y 569.356,Z 923.03,A -85,B 0,C 180,E1 9478.853,E2 9478.853} C_VEL
LIN {X 0,Y 569.243,Z 923.03,A -85,B 0,C 180,E1 9484.619,E2 9484.619} C_VEL
LIN {X 0,Y 569.186,Z 923.03,A -85,B 0,C 180,E1 9489.652,E2 9489.652} C_VEL
LIN {X 0,Y 569.206,Z 923.03,A -85,B 0,C 180,E1 9495.765,E2 9495.765} C_VEL
LIN {X 0,Y 569.166,Z 923.03,A -85,B 0,C 180,E1 9500.416,E2 9500.416} C_VEL
LIN {X 0,Y 569.159,Z 923.03,A -85,B 0,C 180,E1 9506.112,E2 9506.112} C_VEL
LIN {X 0,Y 569.406,Z 923.03,A -85,B 0,C 180,E1 9509.599,E2 9509.599} C_VEL
LIN {X 0,Y 584.009,Z 965.678,A -85,B 0,C 180,E1 9511.36,E2 9511.36} C_VEL
LIN {X 0,Y 585.85,Z 976.394,A -85,B 0,C 180,E1 9511.815,E2 9511.815} C_VEL
LIN {X 0,Y 583.341,Z 1013.481,A -85,B 0,C 180,E1 9513.36,E2 9513.36} C_VEL
LIN {X 0,Y 580.434,Z 1049.152,A -85,B 0,C 180,E1 9515.465,E2 9515.465} C_VEL
LIN {X 0,Y 577.492,Z 1081.171,A -85,B 0,C 180,E1 9518.016,E2 9518.016} C_VEL
LIN {X 0,Y 574.687,Z 1110.525,A -85,B 0,C 180,E1 9521.133,E2 9521.133} C_VEL
LIN {X 0,Y 572.729,Z 1135.404,A -85,B 0,C 180,E1 9524.7,E2 9524.7} C_VEL
LIN {X 0,Y 571.324,Z 1154.048,A -85,B 0,C 180,E1 9528.4,E2 9528.4} C_VEL
LIN {X 0,Y 570.643,Z 1167.6,A -85,B 0,C 180,E1 9532.39,E2 9532.39} C_VEL
LIN {X 0,Y 570.434,Z 1173.971,A -85,B 0,C 180,E1 9535.44,E2 9535.44} C_VEL
LIN {X 0,Y 570.342,Z 1177.159,A -85,B 0,C 180,E1 9538.48,E2 9538.48} C_VEL
LIN {X 0,Y 570.35,Z 1177.161,A -85,B 0,C 180,E1 9541.517,E2 9541.517} C_VEL
LIN {X 0,Y 570.558,Z 1172.789,A -85,B 0,C 180,E1 9545.317,E2 9545.317} C_VEL
LIN {X 0,Y 570.894,Z 1163.241,A -85,B 0,C 180,E1 9549.136,E2 9549.136} C_VEL
LIN {X 0,Y 571.79,Z 1147.802,A -85,B 0,C 180,E1 9552.98,E2 9552.98} C_VEL
LIN {X 0,Y 573.421,Z 1126.781,A -85,B 0,C 180,E1 9556.627,E2 9556.627} C_VEL
LIN {X 0,Y 575.564,Z 1101.983,A -85,B 0,C 180,E1 9559.803,E2 9559.803} C_VEL
LIN {X 0,Y 578.257,Z 1072.226,A -85,B 0,C 180,E1 9562.67,E2 9562.67} C_VEL
LIN {X 0,Y 581.052,Z 1040.045,A -85,B 0,C 180,E1 9564.997,E2 9564.997} C_VEL
LIN {X 0,Y 583.704,Z 1003.344,A -85,B 0,C 180,E1 9566.946,E2 9566.946} C_VEL
LIN {X 0,Y 584.886,Z 971.074,A -85,B 0,C 180,E1 9568.197,E2 9568.197} C_VEL
LIN {X 0,Y 573.581,Z 934.034,A -85,B 0,C 180,E1 9569.826,E2 9569.826} C_VEL
LIN {X 0,Y 569.422,Z 923.03,A -85,B 0,C 180,E1 9570.337,E2 9570.337} C_VEL
LIN {X 0,Y 569.242,Z 923.03,A -85,B 0,C 180,E1 9575.731,E2 9575.731} C_VEL
LIN {X 0,Y 569.066,Z 923.03,A -85,B 0,C 180,E1 9581.995,E2 9581.995} C_VEL
LIN {X 0,Y 569.08,Z 923.03,A -85,B 0,C 180,E1 9588.027,E2 9588.027} C_VEL
LIN {X 0,Y 569.275,Z 923.03,A -85,B 0,C 180,E1 9594.3,E2 9594.3} C_VEL
LIN {X 0,Y 565.213,Z 923.03,A -85,B 0,C 180,E1 9596.024,E2 9596.024} C_VEL
LIN {X 0,Y 561.334,Z 923.03,A -85,B 0,C 180,E1 9597.772,E2 9597.772} C_VEL
LIN {X 0,Y 561.418,Z 923.189,A -85,B 0,C 180,E1 9598.394,E2 9598.394} C_VEL
LIN {X 0,Y 575.288,Z 960.276,A -85,B 0,C 180,E1 9599.932,E2 9599.932} C_VEL
LIN {X 0,Y 579.526,Z 976.308,A -85,B 0,C 180,E1 9600.446,E2 9600.446} C_VEL
LIN {X 0,Y 577.344,Z 1019.799,A -85,B 0,C 180,E1 9601.493,E2 9601.493} C_VEL
LIN {X 0,Y 574.542,Z 1061.235,A -85,B 0,C 180,E1 9603.143,E2 9603.143} C_VEL
LIN {X 0,Y 571.554,Z 1098.871,A -85,B 0,C 180,E1 9605.292,E2 9605.292} C_VEL
LIN {X 0,Y 568.782,Z 1132.289,A -85,B 0,C 180,E1 9607.873,E2 9607.873} C_VEL
LIN {X 0,Y 566.273,Z 1162.195,A -85,B 0,C 180,E1 9610.936,E2 9610.936} C_VEL
LIN {X 0,Y 564.443,Z 1186.831,A -85,B 0,C 180,E1 9614.288,E2 9614.288} C_VEL
LIN {X 0,Y 563.281,Z 1207.031,A -85,B 0,C 180,E1 9618.033,E2 9618.033} C_VEL
LIN {X 0,Y 562.728,Z 1221.375,A -85,B 0,C 180,E1 9621.91,E2 9621.91} C_VEL
LIN {X 0,Y 562.494,Z 1229.227,A -85,B 0,C 180,E1 9625.391,E2 9625.391} C_VEL
LIN {X 0,Y 562.448,Z 1232.64,A -85,B 0,C 180,E1 9628.474,E2 9628.474} C_VEL
LIN {X 0,Y 562.57,Z 1232.698,A -85,B 0,C 180,E1 9631.553,E2 9631.553} C_VEL
LIN {X 0,Y 562.599,Z 1228.159,A -85,B 0,C 180,E1 9635.407,E2 9635.407} C_VEL
LIN {X 0,Y 562.822,Z 1218.218,A -85,B 0,C 180,E1 9639.283,E2 9639.283} C_VEL
LIN {X 0,Y 563.557,Z 1202.274,A -85,B 0,C 180,E1 9643.187,E2 9643.187} C_VEL
LIN {X 0,Y 565.105,Z 1180.547,A -85,B 0,C 180,E1 9646.918,E2 9646.918} C_VEL
LIN {X 0,Y 567.377,Z 1154.134,A -85,B 0,C 180,E1 9650.269,E2 9650.269} C_VEL
LIN {X 0,Y 570.112,Z 1124.338,A -85,B 0,C 180,E1 9653.129,E2 9653.129} C_VEL
LIN {X 0,Y 573.285,Z 1090.391,A -85,B 0,C 180,E1 9655.583,E2 9655.583} C_VEL
LIN {X 0,Y 576.342,Z 1053.424,A -85,B 0,C 180,E1 9657.535,E2 9657.535} C_VEL
LIN {X 0,Y 578.997,Z 1012.764,A -85,B 0,C 180,E1 9658.994,E2 9658.994} C_VEL
LIN {X 0,Y 579.996,Z 973.137,A -85,B 0,C 180,E1 9659.853,E2 9659.853} C_VEL
LIN {X 0,Y 561.476,Z 923.03,A -85,B 0,C 180,E1 9661.603,E2 9661.603} C_VEL
LIN {X 0,Y 561.305,Z 923.03,A -85,B 0,C 180,E1 9666.331,E2 9666.331} C_VEL
LIN {X 0,Y 561.132,Z 923.03,A -85,B 0,C 180,E1 9672.331,E2 9672.331} C_VEL
LIN {X 0,Y 561.132,Z 923.03,A -85,B 0,C 180,E1 9677.685,E2 9677.685} C_VEL
LIN {X 0,Y 561.319,Z 923.03,A -85,B 0,C 180,E1 9683.879,E2 9683.879} C_VEL
LIN {X 0,Y 561.339,Z 923.03,A -85,B 0,C 180,E1 9689.495,E2 9689.495} C_VEL
LIN {X 0,Y 561.495,Z 923.03,A -85,B 0,C 180,E1 9694.497,E2 9694.497} C_VEL
LIN {X 0,Y 561.502,Z 923.03,A -85,B 0,C 180,E1 9700.4,E2 9700.4} C_VEL
LIN {X 0,Y 561.659,Z 923.03,A -85,B 0,C 180,E1 9705.989,E2 9705.989} C_VEL
LIN {X 0,Y 561.973,Z 923.03,A -85,B 0,C 180,E1 9710.717,E2 9710.717} C_VEL
LIN {X 0,Y 562.002,Z 923.03,A -85,B 0,C 180,E1 9713.537,E2 9713.537} C_VEL
LIN {X 0,Y 568.418,Z 952.585,A -85,B 0,C 180,E1 9714.209,E2 9714.209} C_VEL
LIN {X 0,Y 568.258,Z 989.792,A -85,B 0,C 180,E1 9714.9,E2 9714.9} C_VEL
LIN {X 0,Y 567.615,Z 1019.601,A -85,B 0,C 180,E1 9716.09,E2 9716.09} C_VEL
LIN {X 0,Y 566.687,Z 1045.335,A -85,B 0,C 180,E1 9717.805,E2 9717.805} C_VEL
LIN {X 0,Y 565.637,Z 1067.089,A -85,B 0,C 180,E1 9720.002,E2 9720.002} C_VEL
LIN {X 0,Y 564.754,Z 1083.477,A -85,B 0,C 180,E1 9722.494,E2 9722.494} C_VEL
LIN {X 0,Y 564.02,Z 1093.936,A -85,B 0,C 180,E1 9724.997,E2 9724.997} C_VEL
LIN {X 0,Y 563.627,Z 1099.892,A -85,B 0,C 180,E1 9727.705,E2 9727.705} C_VEL
LIN {X 0,Y 563.48,Z 1101.071,A -85,B 0,C 180,E1 9729.261,E2 9729.261} C_VEL
LIN {X 0,Y 563.532,Z 1099.513,A -85,B 0,C 180,E1 9731.84,E2 9731.84} C_VEL
LIN {X 0,Y 563.831,Z 1091.809,A -85,B 0,C 180,E1 9734.912,E2 9734.912} C_VEL
LIN {X 0,Y 564.363,Z 1078.761,A -85,B 0,C 180,E1 9737.669,E2 9737.669} C_VEL
LIN {X 0,Y 565.106,Z 1060.438,A -85,B 0,C 180,E1 9740.14,E2 9740.14} C_VEL
LIN {X 0,Y 566.019,Z 1037.306,A -85,B 0,C 180,E1 9742.241,E2 9742.241} C_VEL
LIN {X 0,Y 566.961,Z 1009.997,A -85,B 0,C 180,E1 9743.86,E2 9743.86} C_VEL
LIN {X 0,Y 567.419,Z 981.744,A -85,B 0,C 180,E1 9744.867,E2 9744.867} C_VEL
LIN {X 0,Y 566.902,Z 947.522,A -85,B 0,C 180,E1 9745.454,E2 9745.454} C_VEL
LIN {X 0,Y 561.664,Z 923.03,A -85,B 0,C 180,E1 9745.961,E2 9745.961} C_VEL
LIN {X 0,Y 561.256,Z 923.03,A -85,B 0,C 180,E1 9752.582,E2 9752.582} C_VEL
LIN {X 0,Y 561.195,Z 923.03,A -85,B 0,C 180,E1 9758.268,E2 9758.268} C_VEL
LIN {X 0,Y 561.11,Z 923.03,A -85,B 0,C 180,E1 9764.445,E2 9764.445} C_VEL
LIN {X 0,Y 561.205,Z 923.03,A -85,B 0,C 180,E1 9769.729,E2 9769.729} C_VEL
LIN {X 0,Y 561.31,Z 923.03,A -85,B 0,C 180,E1 9775.561,E2 9775.561} C_VEL
LIN {X 0,Y 561.431,Z 923.03,A -85,B 0,C 180,E1 9781.01,E2 9781.01} C_VEL
LIN {X 0,Y 561.556,Z 923.03,A -85,B 0,C 180,E1 9786.197,E2 9786.197} C_VEL
LIN {X 0,Y 561.659,Z 923.03,A -85,B 0,C 180,E1 9791.152,E2 9791.152} C_VEL
LIN {X 0,Y 561.721,Z 923.03,A -85,B 0,C 180,E1 9795.976,E2 9795.976} C_VEL
LIN {X 0,Y 561.956,Z 923.03,A -85,B 0,C 180,E1 9800.702,E2 9800.702} C_VEL
LIN {X 0,Y 562.159,Z 923.03,A -85,B 0,C 180,E1 9805.361,E2 9805.361} C_VEL
LIN {X 0,Y 562.372,Z 923.03,A -85,B 0,C 180,E1 9809.986,E2 9809.986} C_VEL
LIN {X 0,Y 562.149,Z 923.03,A -85,B 0,C 180,E1 9816.158,E2 9816.158} C_VEL
LIN {X 0,Y 561.92,Z 923.03,A -85,B 0,C 180,E1 9820.835,E2 9820.835} C_VEL
LIN {X 0,Y 561.792,Z 923.03,A -85,B 0,C 180,E1 9825.588,E2 9825.588} C_VEL
LIN {X 0,Y 561.649,Z 923.03,A -85,B 0,C 180,E1 9830.456,E2 9830.456} C_VEL
LIN {X 0,Y 561.537,Z 923.03,A -85,B 0,C 180,E1 9835.486,E2 9835.486} C_VEL
LIN {X 0,Y 561.444,Z 923.03,A -85,B 0,C 180,E1 9840.736,E2 9840.736} C_VEL
LIN {X 0,Y 561.299,Z 923.03,A -85,B 0,C 180,E1 9846.298,E2 9846.298} C_VEL
LIN {X 0,Y 561.271,Z 923.03,A -85,B 0,C 180,E1 9852.281,E2 9852.281} C_VEL
LIN {X 0,Y 561.239,Z 923.03,A -85,B 0,C 180,E1 9857.69,E2 9857.69} C_VEL
LIN {X 0,Y 561.241,Z 923.03,A -85,B 0,C 180,E1 9863.844,E2 9863.844} C_VEL
LIN {X 0,Y 561.441,Z 923.088,A -85,B 0,C 180,E1 9869.218,E2 9869.218} C_VEL
LIN {X 0,Y 575.457,Z 963.481,A -85,B 0,C 180,E1 9870.891,E2 9870.891} C_VEL
LIN {X 0,Y 578.595,Z 977.622,A -85,B 0,C 180,E1 9871.529,E2 9871.529} C_VEL
LIN {X 0,Y 576.003,Z 1014.254,A -85,B 0,C 180,E1 9873.081,E2 9873.081} C_VEL
LIN {X 0,Y 573.111,Z 1048.659,A -85,B 0,C 180,E1 9875.131,E2 9875.131} C_VEL
LIN {X 0,Y 570.044,Z 1080.539,A -85,B 0,C 180,E1 9877.679,E2 9877.679} C_VEL
LIN {X 0,Y 567.207,Z 1109.327,A -85,B 0,C 180,E1 9880.733,E2 9880.733} C_VEL
LIN {X 0,Y 565.212,Z 1132.584,A -85,B 0,C 180,E1 9884.011,E2 9884.011} C_VEL
LIN {X 0,Y 563.692,Z 1151.538,A -85,B 0,C 180,E1 9887.615,E2 9887.615} C_VEL
LIN {X 0,Y 562.886,Z 1165.748,A -85,B 0,C 180,E1 9891.508,E2 9891.508} C_VEL
LIN {X 0,Y 562.546,Z 1174.314,A -85,B 0,C 180,E1 9895.376,E2 9895.376} C_VEL
LIN {X 0,Y 562.45,Z 1177.536,A -85,B 0,C 180,E1 9898.459,E2 9898.459} C_VEL
LIN {X 0,Y 562.459,Z 1177.553,A -85,B 0,C 180,E1 9901.538,E2 9901.538} C_VEL
LIN {X 0,Y 562.69,Z 1173.171,A -85,B 0,C 180,E1 9905.392,E2 9905.392} C_VEL
LIN {X 0,Y 563.041,Z 1163.587,A -85,B 0,C 180,E1 9909.265,E2 9909.265} C_VEL
LIN {X 0,Y 564.006,Z 1148.101,A -85,B 0,C 180,E1 9913.162,E2 9913.162} C_VEL
LIN {X 0,Y 565.673,Z 1127.975,A -85,B 0,C 180,E1 9916.718,E2 9916.718} C_VEL
LIN {X 0,Y 567.946,Z 1103.125,A -85,B 0,C 180,E1 9919.967,E2 9919.967} C_VEL
LIN {X 0,Y 570.775,Z 1073.472,A -85,B 0,C 180,E1 9922.88,E2 9922.88} C_VEL
LIN {X 0,Y 573.832,Z 1040.031,A -85,B 0,C 180,E1 9925.334,E2 9925.334} C_VEL
LIN {X 0,Y 576.607,Z 1003.093,A -85,B 0,C 180,E1 9927.313,E2 9927.313} C_VEL
LIN {X 0,Y 577.739,Z 972.876,A -85,B 0,C 180,E1 9928.511,E2 9928.511} C_VEL
LIN {X 0,Y 566.811,Z 936.465,A -85,B 0,C 180,E1 9930.187,E2 9930.187} C_VEL
LIN {X 0,Y 561.486,Z 923.03,A -85,B 0,C 180,E1 9930.85,E2 9930.85} C_VEL
LIN {X 0,Y 561.299,Z 923.03,A -85,B 0,C 180,E1 9936.316,E2 9936.316} C_VEL
LIN {X 0,Y 561.126,Z 923.03,A -85,B 0,C 180,E1 9942.316,E2 9942.316} C_VEL
LIN {X 0,Y 561.138,Z 923.03,A -85,B 0,C 180,E1 9947.707,E2 9947.707} C_VEL
LIN {X 0,Y 561.349,Z 923.03,A -85,B 0,C 180,E1 9953.856,E2 9953.856} C_VEL
LIN {X 0,Y 561.334,Z 923.03,A -85,B 0,C 180,E1 9957.772,E2 9957.772} C_VEL
LIN {X 0,Y 562.177,Z 926.313,A -85,B 0,C 180,E1 9958.363,E2 9958.363} C_VEL
LIN {X 0,Y 563.723,Z 934.934,A -85,B 0,C 180,E1 9958.777,E2 9958.777} C_VEL
LIN {X 0,Y 566.019,Z 954.576,A -85,B 0,C 180,E1 9959.287,E2 9959.287} C_VEL
LIN {X 0,Y 572.494,Z 978.629,A -85,B 0,C 180,E1 9960.11,E2 9960.11} C_VEL
LIN {X 0,Y 570.12,Z 1022.061,A -85,B 0,C 180,E1 9961.228,E2 9961.228} C_VEL
LIN {X 0,Y 567.174,Z 1062.055,A -85,B 0,C 180,E1 9962.872,E2 9962.872} C_VEL
LIN {X 0,Y 564.019,Z 1099.623,A -85,B 0,C 180,E1 9965.069,E2 9965.069} C_VEL
LIN {X 0,Y 561.054,Z 1133.595,A -85,B 0,C 180,E1 9967.761,E2 9967.761} C_VEL
LIN {X 0,Y 558.477,Z 1163.095,A -85,B 0,C 180,E1 9970.865,E2 9970.865} C_VEL
LIN {X 0,Y 556.488,Z 1188.671,A -85,B 0,C 180,E1 9974.464,E2 9974.464} C_VEL
LIN {X 0,Y 555.405,Z 1207.086,A -85,B 0,C 180,E1 9977.998,E2 9977.998} C_VEL
LIN {X 0,Y 554.865,Z 1220.89,A -85,B 0,C 180,E1 9981.795,E2 9981.795} C_VEL
LIN {X 0,Y 554.615,Z 1228.801,A -85,B 0,C 180,E1 9985.326,E2 9985.326} C_VEL
LIN {X 0,Y 554.576,Z 1232.245,A -85,B 0,C 180,E1 9988.453,E2 9988.453} C_VEL
LIN {X 0,Y 554.689,Z 1232.312,A -85,B 0,C 180,E1 9991.575,E2 9991.575} C_VEL
LIN {X 0,Y 554.711,Z 1227.779,A -85,B 0,C 180,E1 9995.471,E2 9995.471} C_VEL
LIN {X 0,Y 554.942,Z 1217.764,A -85,B 0,C 180,E1 9999.416,E2 9999.416} C_VEL
LIN {X 0,Y 555.72,Z 1201.739,A -85,B 0,C 180,E1 10003.376,E2 10003.376} C_VEL
LIN {X 0,Y 557.238,Z 1181.249,A -85,B 0,C 180,E1 10006.961,E2 10006.961} C_VEL
LIN {X 0,Y 559.575,Z 1155.117,A -85,B 0,C 180,E1 10010.358,E2 10010.358} C_VEL
LIN {X 0,Y 562.535,Z 1124.508,A -85,B 0,C 180,E1 10013.354,E2 10013.354} C_VEL
LIN {X 0,Y 565.793,Z 1090.887,A -85,B 0,C 180,E1 10015.823,E2 10015.823} C_VEL
LIN {X 0,Y 568.966,Z 1053.871,A -85,B 0,C 180,E1 10017.816,E2 10017.816} C_VEL
LIN {X 0,Y 571.763,Z 1013.517,A -85,B 0,C 180,E1 10019.294,E2 10019.294} C_VEL
LIN {X 0,Y 572.82,Z 974.908,A -85,B 0,C 180,E1 10020.165,E2 10020.165} C_VEL
LIN {X 0,Y 553.517,Z 923.03,A -85,B 0,C 180,E1 10022.034,E2 10022.034} C_VEL
LIN {X 0,Y 553.266,Z 923.03,A -85,B 0,C 180,E1 10027.625,E2 10027.625} C_VEL
LIN {X 0,Y 553.216,Z 923.03,A -85,B 0,C 180,E1 10033.082,E2 10033.082} C_VEL
LIN {X 0,Y 553.248,Z 923.03,A -85,B 0,C 180,E1 10039.043,E2 10039.043} C_VEL
LIN {X 0,Y 553.387,Z 923.03,A -85,B 0,C 180,E1 10045.02,E2 10045.02} C_VEL
LIN {X 0,Y 553.473,Z 923.03,A -85,B 0,C 180,E1 10050.906,E2 10050.906} C_VEL
LIN {X 0,Y 553.58,Z 923.03,A -85,B 0,C 180,E1 10055.831,E2 10055.831} C_VEL
LIN {X 0,Y 553.591,Z 923.03,A -85,B 0,C 180,E1 10060.881,E2 10060.881} C_VEL
LIN {X 0,Y 553.74,Z 923.03,A -85,B 0,C 180,E1 10065.784,E2 10065.784} C_VEL
LIN {X 0,Y 554.05,Z 923.03,A -85,B 0,C 180,E1 10070.583,E2 10070.583} C_VEL
LIN {X 0,Y 554.155,Z 923.775,A -85,B 0,C 180,E1 10073.263,E2 10073.263} C_VEL
LIN {X 0,Y 560.931,Z 953.505,A -85,B 0,C 180,E1 10073.972,E2 10073.972} C_VEL
LIN {X 0,Y 560.74,Z 990.688,A -85,B 0,C 180,E1 10074.674,E2 10074.674} C_VEL
LIN {X 0,Y 560.08,Z 1019.911,A -85,B 0,C 180,E1 10075.844,E2 10075.844} C_VEL
LIN {X 0,Y 559.095,Z 1045.905,A -85,B 0,C 180,E1 10077.581,E2 10077.581} C_VEL
LIN {X 0,Y 557.976,Z 1067.786,A -85,B 0,C 180,E1 10079.808,E2 10079.808} C_VEL
LIN {X 0,Y 557.021,Z 1084.267,A -85,B 0,C 180,E1 10082.334,E2 10082.334} C_VEL
LIN {X 0,Y 556.197,Z 1095.435,A -85,B 0,C 180,E1 10085.067,E2 10085.067} C_VEL
LIN {X 0,Y 555.781,Z 1101.07,A -85,B 0,C 180,E1 10087.815,E2 10087.815} C_VEL
LIN {X 0,Y 555.645,Z 1102.036,A -85,B 0,C 180,E1 10089.393,E2 10089.393} C_VEL
LIN {X 0,Y 555.674,Z 1100.582,A -85,B 0,C 180,E1 10091.726,E2 10091.726} C_VEL
LIN {X 0,Y 555.98,Z 1093.443,A -85,B 0,C 180,E1 10094.736,E2 10094.736} C_VEL
LIN {X 0,Y 556.5,Z 1080.549,A -85,B 0,C 180,E1 10097.574,E2 10097.574} C_VEL
LIN {X 0,Y 557.235,Z 1063.202,A -85,B 0,C 180,E1 10100.023,E2 10100.023} C_VEL
LIN {X 0,Y 558.152,Z 1040.613,A -85,B 0,C 180,E1 10102.17,E2 10102.17} C_VEL
LIN {X 0,Y 559.163,Z 1013.868,A -85,B 0,C 180,E1 10103.856,E2 10103.856} C_VEL
LIN {X 0,Y 559.697,Z 984.1,A -85,B 0,C 180,E1 10104.981,E2 10104.981} C_VEL
LIN {X 0,Y 559.076,Z 947.975,A -85,B 0,C 180,E1 10105.631,E2 10105.631} C_VEL
LIN {X 0,Y 553.724,Z 923.03,A -85,B 0,C 180,E1 10106.173,E2 10106.173} C_VEL
LIN {X 0,Y 553.314,Z 923.03,A -85,B 0,C 180,E1 10112.138,E2 10112.138} C_VEL
LIN {X 0,Y 553.263,Z 923.03,A -85,B 0,C 180,E1 10117.606,E2 10117.606} C_VEL
LIN {X 0,Y 553.204,Z 923.03,A -85,B 0,C 180,E1 10123.072,E2 10123.072} C_VEL
LIN {X 0,Y 553.277,Z 923.03,A -85,B 0,C 180,E1 10129.03,E2 10129.03} C_VEL
LIN {X 0,Y 553.355,Z 923.03,A -85,B 0,C 180,E1 10135.011,E2 10135.011} C_VEL
LIN {X 0,Y 553.527,Z 923.03,A -85,B 0,C 180,E1 10140.881,E2 10140.881} C_VEL
LIN {X 0,Y 553.629,Z 923.03,A -85,B 0,C 180,E1 10145.819,E2 10145.819} C_VEL
LIN {X 0,Y 553.774,Z 923.03,A -85,B 0,C 180,E1 10150.873,E2 10150.873} C_VEL
LIN {X 0,Y 553.832,Z 923.03,A -85,B 0,C 180,E1 10155.772,E2 10155.772} C_VEL
LIN {X 0,Y 554.034,Z 923.03,A -85,B 0,C 180,E1 10160.568,E2 10160.568} C_VEL
LIN {X 0,Y 554.257,Z 923.03,A -85,B 0,C 180,E1 10165.295,E2 10165.295} C_VEL
LIN {X 0,Y 554.495,Z 923.03,A -85,B 0,C 180,E1 10169.986,E2 10169.986} C_VEL
LIN {X 0,Y 554.233,Z 923.03,A -85,B 0,C 180,E1 10176.247,E2 10176.247} C_VEL
LIN {X 0,Y 554.012,Z 923.03,A -85,B 0,C 180,E1 10180.992,E2 10180.992} C_VEL
LIN {X 0,Y 553.863,Z 923.03,A -85,B 0,C 180,E1 10185.817,E2 10185.817} C_VEL
LIN {X 0,Y 553.699,Z 923.03,A -85,B 0,C 180,E1 10190.763,E2 10190.763} C_VEL
LIN {X 0,Y 553.58,Z 923.03,A -85,B 0,C 180,E1 10195.879,E2 10195.879} C_VEL
LIN {X 0,Y 553.466,Z 923.03,A -85,B 0,C 180,E1 10201.229,E2 10201.229} C_VEL
LIN {X 0,Y 553.309,Z 923.03,A -85,B 0,C 180,E1 10206.908,E2 10206.908} C_VEL
LIN {X 0,Y 553.381,Z 923.03,A -85,B 0,C 180,E1 10213.028,E2 10213.028} C_VEL
LIN {X 0,Y 553.304,Z 923.03,A -85,B 0,C 180,E1 10219.044,E2 10219.044} C_VEL
LIN {X 0,Y 553.325,Z 923.03,A -85,B 0,C 180,E1 10225.004,E2 10225.004} C_VEL
LIN {X 0,Y 553.476,Z 923.094,A -85,B 0,C 180,E1 10228.813,E2 10228.813} C_VEL
LIN {X 0,Y 567.702,Z 963.669,A -85,B 0,C 180,E1 10230.527,E2 10230.527} C_VEL
LIN {X 0,Y 571.4,Z 978.166,A -85,B 0,C 180,E1 10231.215,E2 10231.215} C_VEL
LIN {X 0,Y 568.547,Z 1016.559,A -85,B 0,C 180,E1 10232.88,E2 10232.88} C_VEL
LIN {X 0,Y 565.425,Z 1051.853,A -85,B 0,C 180,E1 10235.052,E2 10235.052} C_VEL
LIN {X 0,Y 562.122,Z 1084.754,A -85,B 0,C 180,E1 10237.787,E2 10237.787} C_VEL
LIN {X 0,Y 559.107,Z 1114.117,A -85,B 0,C 180,E1 10241.074,E2 10241.074} C_VEL
LIN {X 0,Y 557.057,Z 1137.815,A -85,B 0,C 180,E1 10244.662,E2 10244.662} C_VEL
LIN {X 0,Y 555.68,Z 1154.744,A -85,B 0,C 180,E1 10248.136,E2 10248.136} C_VEL
LIN {X 0,Y 554.917,Z 1168.201,A -85,B 0,C 180,E1 10252.173,E2 10252.173} C_VEL
LIN {X 0,Y 554.594,Z 1175.797,A -85,B 0,C 180,E1 10256.092,E2 10256.092} C_VEL
LIN {X 0,Y 554.465,Z 1178.356,A -85,B 0,C 180,E1 10259.998,E2 10259.998} C_VEL
LIN {X 0,Y 554.599,Z 1176.763,A -85,B 0,C 180,E1 10263.122,E2 10263.122} C_VEL
LIN {X 0,Y 554.947,Z 1170.801,A -85,B 0,C 180,E1 10266.842,E2 10266.842} C_VEL
LIN {X 0,Y 555.566,Z 1158.464,A -85,B 0,C 180,E1 10270.974,E2 10270.974} C_VEL
LIN {X 0,Y 556.855,Z 1141.394,A -85,B 0,C 180,E1 10274.736,E2 10274.736} C_VEL
LIN {X 0,Y 558.738,Z 1120.259,A -85,B 0,C 180,E1 10278.119,E2 10278.119} C_VEL
LIN {X 0,Y 561.332,Z 1094.234,A -85,B 0,C 180,E1 10281.245,E2 10281.245} C_VEL
LIN {X 0,Y 564.322,Z 1064.608,A -85,B 0,C 180,E1 10283.941,E2 10283.941} C_VEL
LIN {X 0,Y 567.459,Z 1030.352,A -85,B 0,C 180,E1 10286.275,E2 10286.275} C_VEL
LIN {X 0,Y 570.262,Z 993.113,A -85,B 0,C 180,E1 10288.109,E2 10288.109} C_VEL
LIN {X 0,Y 570.641,Z 974.86,A -85,B 0,C 180,E1 10288.833,E2 10288.833} C_VEL
LIN {X 0,Y 560.372,Z 939.781,A -85,B 0,C 180,E1 10290.525,E2 10290.525} C_VEL
LIN {X 0,Y 553.583,Z 923.03,A -85,B 0,C 180,E1 10291.404,E2 10291.404} C_VEL
LIN {X 0,Y 553.294,Z 923.03,A -85,B 0,C 180,E1 10296.928,E2 10296.928} C_VEL
LIN {X 0,Y 553.226,Z 923.03,A -85,B 0,C 180,E1 10303.065,E2 10303.065} C_VEL
LIN {X 0,Y 553.245,Z 923.03,A -85,B 0,C 180,E1 10309.064,E2 10309.064} C_VEL
LIN {X 0,Y 553.399,Z 923.03,A -85,B 0,C 180,E1 10315.031,E2 10315.031} C_VEL
LIN {X 0,Y 553.518,Z 923.728,A -85,B 0,C 180,E1 10317.841,E2 10317.841} C_VEL
LIN {X 0,Y 566.019,Z 954.576,A -85,B 0,C 180,E1 10319.287,E2 10319.287} C_VEL
LIN {X 0,Y 567.783,Z 968.301,A -85,B 0,C 180,E1 10319.641,E2 10319.641} C_VEL
LIN {X 0,Y 565.105,Z 989.477,A -85,B 0,C 180,E1 10319.951,E2 10319.951} C_VEL
LIN {X 0,Y 562.267,Z 1032.777,A -85,B 0,C 180,E1 10321.253,E2 10321.253} C_VEL
LIN {X 0,Y 558.894,Z 1073.5,A -85,B 0,C 180,E1 10323.151,E2 10323.151} C_VEL
LIN {X 0,Y 555.714,Z 1109.402,A -85,B 0,C 180,E1 10325.493,E2 10325.493} C_VEL
LIN {X 0,Y 552.752,Z 1141.328,A -85,B 0,C 180,E1 10328.271,E2 10328.271} C_VEL
LIN {X 0,Y 550.142,Z 1169.646,A -85,B 0,C 180,E1 10331.52,E2 10331.52} C_VEL
LIN {X 0,Y 548.345,Z 1193.13,A -85,B 0,C 180,E1 10335.124,E2 10335.124} C_VEL
LIN {X 0,Y 547.342,Z 1210.859,A -85,B 0,C 180,E1 10338.872,E2 10338.872} C_VEL
LIN {X 0,Y 546.838,Z 1223.571,A -85,B 0,C 180,E1 10342.871,E2 10342.871} C_VEL
LIN {X 0,Y 546.721,Z 1230.532,A -85,B 0,C 180,E1 10346.845,E2 10346.845} C_VEL
LIN {X 0,Y 546.712,Z 1232.331,A -85,B 0,C 180,E1 10350.014,E2 10350.014} C_VEL
LIN {X 0,Y 546.728,Z 1229.807,A -85,B 0,C 180,E1 10353.976,E2 10353.976} C_VEL
LIN {X 0,Y 546.943,Z 1221.97,A -85,B 0,C 180,E1 10357.954,E2 10357.954} C_VEL
LIN {X 0,Y 547.531,Z 1208.148,A -85,B 0,C 180,E1 10362.024,E2 10362.024} C_VEL
LIN {X 0,Y 548.888,Z 1188.163,A -85,B 0,C 180,E1 10365.993,E2 10365.993} C_VEL
LIN {X 0,Y 550.961,Z 1164.446,A -85,B 0,C 180,E1 10369.436,E2 10369.436} C_VEL
LIN {X 0,Y 553.929,Z 1134.682,A -85,B 0,C 180,E1 10372.677,E2 10372.677} C_VEL
LIN {X 0,Y 557.155,Z 1102.64,A -85,B 0,C 180,E1 10375.308,E2 10375.308} C_VEL
LIN {X 0,Y 560.498,Z 1066.536,A -85,B 0,C 180,E1 10377.509,E2 10377.509} C_VEL
LIN {X 0,Y 563.626,Z 1028.572,A -85,B 0,C 180,E1 10379.134,E2 10379.134} C_VEL
LIN {X 0,Y 565.869,Z 989.367,A -85,B 0,C 180,E1 10380.212,E2 10380.212} C_VEL
LIN {X 0,Y 565.51,Z 976.378,A -85,B 0,C 180,E1 10380.49,E2 10380.49} C_VEL
LIN {X 0,Y 545.576,Z 923.03,A -85,B 0,C 180,E1 10382.435,E2 10382.435} C_VEL
LIN {X 0,Y 545.395,Z 923.03,A -85,B 0,C 180,E1 10387.57,E2 10387.57} C_VEL
LIN {X 0,Y 545.274,Z 923.03,A -85,B 0,C 180,E1 10393.904,E2 10393.904} C_VEL
LIN {X 0,Y 545.362,Z 923.03,A -85,B 0,C 180,E1 10400.412,E2 10400.412} C_VEL
LIN {X 0,Y 545.421,Z 923.03,A -85,B 0,C 180,E1 10406.353,E2 10406.353} C_VEL
LIN {X 0,Y 545.598,Z 923.03,A -85,B 0,C 180,E1 10412.429,E2 10412.429} C_VEL
LIN {X 0,Y 545.663,Z 923.03,A -85,B 0,C 180,E1 10417.19,E2 10417.19} C_VEL
LIN {X 0,Y 545.687,Z 923.03,A -85,B 0,C 180,E1 10422.267,E2 10422.267} C_VEL
LIN {X 0,Y 545.901,Z 923.03,A -85,B 0,C 180,E1 10427.208,E2 10427.208} C_VEL
LIN {X 0,Y 546.252,Z 923.03,A -85,B 0,C 180,E1 10432.937,E2 10432.937} C_VEL
LIN {X 0,Y 553.454,Z 955.069,A -85,B 0,C 180,E1 10433.732,E2 10433.732} C_VEL
LIN {X 0,Y 553.199,Z 992.522,A -85,B 0,C 180,E1 10434.466,E2 10434.466} C_VEL
LIN {X 0,Y 552.532,Z 1021.968,A -85,B 0,C 180,E1 10435.688,E2 10435.688} C_VEL
LIN {X 0,Y 551.472,Z 1047.666,A -85,B 0,C 180,E1 10437.45,E2 10437.45} C_VEL
LIN {X 0,Y 550.349,Z 1068.539,A -85,B 0,C 180,E1 10439.608,E2 10439.608} C_VEL
LIN {X 0,Y 549.322,Z 1085.098,A -85,B 0,C 180,E1 10442.169,E2 10442.169} C_VEL
LIN {X 0,Y 548.442,Z 1095.693,A -85,B 0,C 180,E1 10444.743,E2 10444.743} C_VEL
LIN {X 0,Y 548.084,Z 1100.897,A -85,B 0,C 180,E1 10446.932,E2 10446.932} C_VEL
LIN {X 0,Y 547.812,Z 1103.002,A -85,B 0,C 180,E1 10449.528,E2 10449.528} C_VEL
LIN {X 0,Y 547.858,Z 1101.283,A -85,B 0,C 180,E1 10451.896,E2 10451.896} C_VEL
LIN {X 0,Y 548.14,Z 1094.237,A -85,B 0,C 180,E1 10454.796,E2 10454.796} C_VEL
LIN {X 0,Y 548.672,Z 1081.431,A -85,B 0,C 180,E1 10457.637,E2 10457.637} C_VEL
LIN {X 0,Y 549.407,Z 1064.532,A -85,B 0,C 180,E1 10460.061,E2 10460.061} C_VEL
LIN {X 0,Y 550.389,Z 1041.495,A -85,B 0,C 180,E1 10462.287,E2 10462.287} C_VEL
LIN {X 0,Y 551.438,Z 1014.496,A -85,B 0,C 180,E1 10464.008,E2 10464.008} C_VEL
LIN {X 0,Y 551.993,Z 985.026,A -85,B 0,C 180,E1 10465.136,E2 10465.136} C_VEL
LIN {X 0,Y 551.288,Z 948.487,A -85,B 0,C 180,E1 10465.808,E2 10465.808} C_VEL
LIN {X 0,Y 545.778,Z 923.03,A -85,B 0,C 180,E1 10466.364,E2 10466.364} C_VEL
LIN {X 0,Y 545.406,Z 923.03,A -85,B 0,C 180,E1 10471.765,E2 10471.765} C_VEL
LIN {X 0,Y 545.394,Z 923.03,A -85,B 0,C 180,E1 10477.559,E2 10477.559} C_VEL
LIN {X 0,Y 545.27,Z 923.03,A -85,B 0,C 180,E1 10483.887,E2 10483.887} C_VEL
LIN {X 0,Y 545.384,Z 923.03,A -85,B 0,C 180,E1 10490.398,E2 10490.398} C_VEL
LIN {X 0,Y 545.396,Z 923.03,A -85,B 0,C 180,E1 10496.336,E2 10496.336} C_VEL
LIN {X 0,Y 545.675,Z 923.03,A -85,B 0,C 180,E1 10502.397,E2 10502.397} C_VEL
LIN {X 0,Y 545.696,Z 923.03,A -85,B 0,C 180,E1 10507.177,E2 10507.177} C_VEL
LIN {X 0,Y 545.867,Z 923.03,A -85,B 0,C 180,E1 10512.259,E2 10512.259} C_VEL
LIN {X 0,Y 545.936,Z 923.03,A -85,B 0,C 180,E1 10517.194,E2 10517.194} C_VEL
LIN {X 0,Y 546.232,Z 923.03,A -85,B 0,C 180,E1 10522.036,E2 10522.036} C_VEL
LIN {X 0,Y 546.474,Z 923.03,A -85,B 0,C 180,E1 10526.816,E2 10526.816} C_VEL
LIN {X 0,Y 546.503,Z 923.03,A -85,B 0,C 180,E1 10531.57,E2 10531.57} C_VEL
LIN {X 0,Y 546.328,Z 923.03,A -85,B 0,C 180,E1 10536.337,E2 10536.337} C_VEL
LIN {X 0,Y 546.088,Z 923.03,A -85,B 0,C 180,E1 10541.153,E2 10541.153} C_VEL
LIN {X 0,Y 545.944,Z 923.03,A -85,B 0,C 180,E1 10546.052,E2 10546.052} C_VEL
LIN {X 0,Y 545.766,Z 923.03,A -85,B 0,C 180,E1 10551.079,E2 10551.079} C_VEL
LIN {X 0,Y 545.631,Z 923.03,A -85,B 0,C 180,E1 10556.284,E2 10556.284} C_VEL
LIN {X 0,Y 545.53,Z 923.03,A -85,B 0,C 180,E1 10561.736,E2 10561.736} C_VEL
LIN {X 0,Y 545.403,Z 923.03,A -85,B 0,C 180,E1 10567.534,E2 10567.534} C_VEL
LIN {X 0,Y 545.422,Z 923.03,A -85,B 0,C 180,E1 10573.916,E2 10573.916} C_VEL
LIN {X 0,Y 545.364,Z 923.03,A -85,B 0,C 180,E1 10580.408,E2 10580.408} C_VEL
LIN {X 0,Y 545.372,Z 923.03,A -85,B 0,C 180,E1 10586.346,E2 10586.346} C_VEL
LIN {X 0,Y 545.553,Z 923.648,A -85,B 0,C 180,E1 10588.411,E2 10588.411} C_VEL
LIN {X 0,Y 560.165,Z 964.753,A -85,B 0,C 180,E1 10590.199,E2 10590.199} C_VEL
LIN {X 0,Y 564.033,Z 981.321,A -85,B 0,C 180,E1 10590.99,E2 10590.99} C_VEL
LIN {X 0,Y 560.97,Z 1020.195,A -85,B 0,C 180,E1 10592.744,E2 10592.744} C_VEL
LIN {X 0,Y 557.62,Z 1056.049,A -85,B 0,C 180,E1 10595.048,E2 10595.048} C_VEL
LIN {X 0,Y 554.158,Z 1089.1,A -85,B 0,C 180,E1 10597.941,E2 10597.941} C_VEL
LIN {X 0,Y 551.323,Z 1115.733,A -85,B 0,C 180,E1 10601.034,E2 10601.034} C_VEL
LIN {X 0,Y 549.243,Z 1138.623,A -85,B 0,C 180,E1 10604.575,E2 10604.575} C_VEL
LIN {X 0,Y 547.747,Z 1156.674,A -85,B 0,C 180,E1 10608.413,E2 10608.413} C_VEL
LIN {X 0,Y 547.067,Z 1168.49,A -85,B 0,C 180,E1 10612.06,E2 10612.06} C_VEL
LIN {X 0,Y 546.725,Z 1176.151,A -85,B 0,C 180,E1 10616.036,E2 10616.036} C_VEL
LIN {X 0,Y 546.576,Z 1178.747,A -85,B 0,C 180,E1 10619.998,E2 10619.998} C_VEL
LIN {X 0,Y 546.711,Z 1177.168,A -85,B 0,C 180,E1 10623.167,E2 10623.167} C_VEL
LIN {X 0,Y 547.104,Z 1170.73,A -85,B 0,C 180,E1 10627.138,E2 10627.138} C_VEL
LIN {X 0,Y 547.767,Z 1158.845,A -85,B 0,C 180,E1 10631.132,E2 10631.132} C_VEL
LIN {X 0,Y 549.115,Z 1141.977,A -85,B 0,C 180,E1 10634.905,E2 10634.905} C_VEL
LIN {X 0,Y 551.149,Z 1120.568,A -85,B 0,C 180,E1 10638.377,E2 10638.377} C_VEL
LIN {X 0,Y 553.911,Z 1094.065,A -85,B 0,C 180,E1 10641.592,E2 10641.592} C_VEL
LIN {X 0,Y 557.197,Z 1062.865,A -85,B 0,C 180,E1 10644.432,E2 10644.432} C_VEL
LIN {X 0,Y 560.614,Z 1027.166,A -85,B 0,C 180,E1 10646.837,E2 10646.837} C_VEL
LIN {X 0,Y 563.676,Z 987.273,A -85,B 0,C 180,E1 10648.74,E2 10648.74} C_VEL
LIN {X 0,Y 563.627,Z 976.759,A -85,B 0,C 180,E1 10649.172,E2 10649.172} C_VEL
LIN {X 0,Y 553.879,Z 942.806,A -85,B 0,C 180,E1 10650.884,E2 10650.884} C_VEL
LIN {X 0,Y 545.647,Z 923.03,A -85,B 0,C 180,E1 10652.006,E2 10652.006} C_VEL
LIN {X 0,Y 545.37,Z 923.03,A -85,B 0,C 180,E1 10657.556,E2 10657.556} C_VEL
LIN {X 0,Y 545.282,Z 923.03,A -85,B 0,C 180,E1 10663.929,E2 10663.929} C_VEL
LIN {X 0,Y 545.348,Z 923.03,A -85,B 0,C 180,E1 10670.431,E2 10670.431} C_VEL
LIN {X 0,Y 545.432,Z 923.03,A -85,B 0,C 180,E1 10676.372,E2 10676.372} C_VEL
LIN {X 0,Y 545.492,Z 923.03,A -85,B 0,C 180,E1 10677.189,E2 10677.189} C_VEL
LIN {X 0,Y 559.837,Z 958.331,A -85,B 0,C 180,E1 10678.967,E2 10678.967} C_VEL
LIN {X 0,Y 565.531,Z 980.503,A -85,B 0,C 180,E1 10679.755,E2 10679.755} C_VEL
LIN {X 0,Y 565.105,Z 989.477,A -85,B 0,C 180,E1 10679.951,E2 10679.951} C_VEL
LIN {X 0,Y 560.409,Z 1006.321,A -85,B 0,C 180,E1 10680.169,E2 10680.169} C_VEL
LIN {X 0,Y 556.113,Z 1020.812,A -85,B 0,C 180,E1 10680.448,E2 10680.448} C_VEL
LIN {X 0,Y 555.933,Z 1022.824,A -85,B 0,C 180,E1 10680.52,E2 10680.52} C_VEL
LIN {X 0,Y 552.727,Z 1062.172,A -85,B 0,C 180,E1 10682.213,E2 10682.213} C_VEL
LIN {X 0,Y 549.263,Z 1099.151,A -85,B 0,C 180,E1 10684.45,E2 10684.45} C_VEL
LIN {X 0,Y 545.892,Z 1133.06,A -85,B 0,C 180,E1 10687.216,E2 10687.216} C_VEL
LIN {X 0,Y 542.971,Z 1163.331,A -85,B 0,C 180,E1 10690.507,E2 10690.507} C_VEL
LIN {X 0,Y 540.837,Z 1188.276,A -85,B 0,C 180,E1 10694.151,E2 10694.151} C_VEL
LIN {X 0,Y 539.648,Z 1207.061,A -85,B 0,C 180,E1 10697.893,E2 10697.893} C_VEL
LIN {X 0,Y 539.049,Z 1221.058,A -85,B 0,C 180,E1 10701.958,E2 10701.958} C_VEL
LIN {X 0,Y 538.863,Z 1229.186,A -85,B 0,C 180,E1 10705.994,E2 10705.994} C_VEL
LIN {X 0,Y 538.831,Z 1231.939,A -85,B 0,C 180,E1 10710.014,E2 10710.014} C_VEL
LIN {X 0,Y 538.848,Z 1229.404,A -85,B 0,C 180,E1 10714.034,E2 10714.034} C_VEL
LIN {X 0,Y 539.053,Z 1221.52,A -85,B 0,C 180,E1 10718.071,E2 10718.071} C_VEL
LIN {X 0,Y 539.641,Z 1208.2,A -85,B 0,C 180,E1 10722.054,E2 10722.054} C_VEL
LIN {X 0,Y 541.019,Z 1188.552,A -85,B 0,C 180,E1 10726.053,E2 10726.053} C_VEL
LIN {X 0,Y 543.31,Z 1163.598,A -85,B 0,C 180,E1 10729.721,E2 10729.721} C_VEL
LIN {X 0,Y 546.295,Z 1134.725,A -85,B 0,C 180,E1 10732.904,E2 10732.904} C_VEL
LIN {X 0,Y 549.802,Z 1101.362,A -85,B 0,C 180,E1 10735.665,E2 10735.665} C_VEL
LIN {X 0,Y 553.297,Z 1064.802,A -85,B 0,C 180,E1 10737.898,E2 10737.898} C_VEL
LIN {X 0,Y 556.553,Z 1025.728,A -85,B 0,C 180,E1 10739.562,E2 10739.562} C_VEL
LIN {X 0,Y 559.001,Z 984.33,A -85,B 0,C 180,E1 10740.66,E2 10740.66} C_VEL
LIN {X 0,Y 557.675,Z 976.254,A -85,B 0,C 180,E1 10740.876,E2 10740.876} C_VEL
LIN {X 0,Y 537.628,Z 923.03,A -85,B 0,C 180,E1 10742.877,E2 10742.877} C_VEL
LIN {X 0,Y 537.45,Z 923.03,A -85,B 0,C 180,E1 10748.224,E2 10748.224} C_VEL
LIN {X 0,Y 537.306,Z 923.03,A -85,B 0,C 180,E1 10754.69,E2 10754.69} C_VEL
LIN {X 0,Y 537.373,Z 923.03,A -85,B 0,C 180,E1 10759.704,E2 10759.704} C_VEL
LIN {X 0,Y 537.471,Z 923.03,A -85,B 0,C 180,E1 10765.787,E2 10765.787} C_VEL
LIN {X 0,Y 537.571,Z 923.03,A -85,B 0,C 180,E1 10771.456,E2 10771.456} C_VEL
LIN {X 0,Y 537.741,Z 923.03,A -85,B 0,C 180,E1 10776.835,E2 10776.835} C_VEL
LIN {X 0,Y 537.781,Z 923.03,A -85,B 0,C 180,E1 10782.846,E2 10782.846} C_VEL
LIN {X 0,Y 538.124,Z 923.03,A -85,B 0,C 180,E1 10788.666,E2 10788.666} C_VEL
LIN {X 0,Y 538.366,Z 923.767,A -85,B 0,C 180,E1 10792.633,E2 10792.633} C_VEL
LIN {X 0,Y 545.953,Z 954.868,A -85,B 0,C 180,E1 10793.453,E2 10793.453} C_VEL
LIN {X 0,Y 545.779,Z 992.512,A -85,B 0,C 180,E1 10794.189,E2 10794.189} C_VEL
LIN {X 0,Y 545.016,Z 1022.462,A -85,B 0,C 180,E1 10795.43,E2 10795.43} C_VEL
LIN {X 0,Y 543.902,Z 1048.257,A -85,B 0,C 180,E1 10797.215,E2 10797.215} C_VEL
LIN {X 0,Y 542.724,Z 1069.29,A -85,B 0,C 180,E1 10799.403,E2 10799.403} C_VEL
LIN {X 0,Y 541.6,Z 1085.959,A -85,B 0,C 180,E1 10802,E2 10802} C_VEL
LIN {X 0,Y 540.629,Z 1097.248,A -85,B 0,C 180,E1 10804.812,E2 10804.812} C_VEL
LIN {X 0,Y 540.238,Z 1102.151,A -85,B 0,C 180,E1 10807.033,E2 10807.033} C_VEL
LIN {X 0,Y 539.978,Z 1103.968,A -85,B 0,C 180,E1 10809.668,E2 10809.668} C_VEL
LIN {X 0,Y 540.023,Z 1101.728,A -85,B 0,C 180,E1 10812.183,E2 10812.183} C_VEL
LIN {X 0,Y 540.342,Z 1094.483,A -85,B 0,C 180,E1 10815.015,E2 10815.015} C_VEL
LIN {X 0,Y 540.944,Z 1081.214,A -85,B 0,C 180,E1 10817.897,E2 10817.897} C_VEL
LIN {X 0,Y 541.776,Z 1062.581,A -85,B 0,C 180,E1 10820.478,E2 10820.478} C_VEL
LIN {X 0,Y 542.741,Z 1039.744,A -85,B 0,C 180,E1 10822.619,E2 10822.619} C_VEL
LIN {X 0,Y 543.74,Z 1013.651,A -85,B 0,C 180,E1 10824.237,E2 10824.237} C_VEL
LIN {X 0,Y 544.299,Z 984.942,A -85,B 0,C 180,E1 10825.324,E2 10825.324} C_VEL
LIN {X 0,Y 543.611,Z 949.587,A -85,B 0,C 180,E1 10825.976,E2 10825.976} C_VEL
LIN {X 0,Y 537.834,Z 923.03,A -85,B 0,C 180,E1 10826.616,E2 10826.616} C_VEL
LIN {X 0,Y 537.446,Z 923.03,A -85,B 0,C 180,E1 10832.472,E2 10832.472} C_VEL
LIN {X 0,Y 537.46,Z 923.03,A -85,B 0,C 180,E1 10838.212,E2 10838.212} C_VEL
LIN {X 0,Y 537.301,Z 923.03,A -85,B 0,C 180,E1 10844.678,E2 10844.678} C_VEL
LIN {X 0,Y 537.394,Z 923.03,A -85,B 0,C 180,E1 10849.69,E2 10849.69} C_VEL
LIN {X 0,Y 537.448,Z 923.03,A -85,B 0,C 180,E1 10855.77,E2 10855.77} C_VEL
LIN {X 0,Y 537.653,Z 923.03,A -85,B 0,C 180,E1 10861.445,E2 10861.445} C_VEL
LIN {X 0,Y 537.779,Z 923.03,A -85,B 0,C 180,E1 10866.822,E2 10866.822} C_VEL
LIN {X 0,Y 537.926,Z 923.03,A -85,B 0,C 180,E1 10872.771,E2 10872.771} C_VEL
LIN {X 0,Y 538.132,Z 923.03,A -85,B 0,C 180,E1 10878.651,E2 10878.651} C_VEL
LIN {X 0,Y 538.37,Z 923.03,A -85,B 0,C 180,E1 10883.54,E2 10883.54} C_VEL
LIN {X 0,Y 538.541,Z 923.03,A -85,B 0,C 180,E1 10888.378,E2 10888.378} C_VEL
LIN {X 0,Y 538.463,Z 923.03,A -85,B 0,C 180,E1 10893.203,E2 10893.203} C_VEL
LIN {X 0,Y 538.317,Z 923.03,A -85,B 0,C 180,E1 10898.053,E2 10898.053} C_VEL
LIN {X 0,Y 538.122,Z 923.03,A -85,B 0,C 180,E1 10902.966,E2 10902.966} C_VEL
LIN {X 0,Y 537.996,Z 923.03,A -85,B 0,C 180,E1 10907.98,E2 10907.98} C_VEL
LIN {X 0,Y 537.788,Z 923.03,A -85,B 0,C 180,E1 10913.147,E2 10913.147} C_VEL
LIN {X 0,Y 537.63,Z 923.03,A -85,B 0,C 180,E1 10919.386,E2 10919.386} C_VEL
LIN {X 0,Y 537.501,Z 923.03,A -85,B 0,C 180,E1 10925.381,E2 10925.381} C_VEL
LIN {X 0,Y 537.424,Z 923.03,A -85,B 0,C 180,E1 10930.606,E2 10930.606} C_VEL
LIN {X 0,Y 537.427,Z 923.03,A -85,B 0,C 180,E1 10936.948,E2 10936.948} C_VEL
LIN {X 0,Y 537.428,Z 923.03,A -85,B 0,C 180,E1 10941.902,E2 10941.902} C_VEL
LIN {X 0,Y 537.557,Z 923.03,A -85,B 0,C 180,E1 10947.967,E2 10947.967} C_VEL
LIN {X 0,Y 552.41,Z 965.257,A -85,B 0,C 180,E1 10949.835,E2 10949.835} C_VEL
LIN {X 0,Y 556.743,Z 982.797,A -85,B 0,C 180,E1 10950.701,E2 10950.701} C_VEL
LIN {X 0,Y 553.475,Z 1022.668,A -85,B 0,C 180,E1 10952.556,E2 10952.556} C_VEL
LIN {X 0,Y 549.834,Z 1058.991,A -85,B 0,C 180,E1 10954.969,E2 10954.969} C_VEL
LIN {X 0,Y 546.507,Z 1090.22,A -85,B 0,C 180,E1 10957.772,E2 10957.772} C_VEL
LIN {X 0,Y 543.529,Z 1117.485,A -85,B 0,C 180,E1 10961.016,E2 10961.016} C_VEL
LIN {X 0,Y 541.46,Z 1139.276,A -85,B 0,C 180,E1 10964.461,E2 10964.461} C_VEL
LIN {X 0,Y 539.941,Z 1157.029,A -85,B 0,C 180,E1 10968.289,E2 10968.289} C_VEL
LIN {X 0,Y 539.206,Z 1168.768,A -85,B 0,C 180,E1 10971.943,E2 10971.943} C_VEL
LIN {X 0,Y 538.84,Z 1176.5,A -85,B 0,C 180,E1 10975.978,E2 10975.978} C_VEL
LIN {X 0,Y 538.694,Z 1179.14,A -85,B 0,C 180,E1 10979.998,E2 10979.998} C_VEL
LIN {X 0,Y 538.823,Z 1177.58,A -85,B 0,C 180,E1 10983.214,E2 10983.214} C_VEL
LIN {X 0,Y 539.235,Z 1171.147,A -85,B 0,C 180,E1 10987.243,E2 10987.243} C_VEL
LIN {X 0,Y 539.968,Z 1159.253,A -85,B 0,C 180,E1 10991.295,E2 10991.295} C_VEL
LIN {X 0,Y 541.443,Z 1141.846,A -85,B 0,C 180,E1 10995.221,E2 10995.221} C_VEL
LIN {X 0,Y 543.692,Z 1119.643,A -85,B 0,C 180,E1 10998.823,E2 10998.823} C_VEL
LIN {X 0,Y 546.715,Z 1092.321,A -85,B 0,C 180,E1 11002.121,E2 11002.121} C_VEL
LIN {X 0,Y 550.24,Z 1060.568,A -85,B 0,C 180,E1 11004.987,E2 11004.987} C_VEL
LIN {X 0,Y 553.874,Z 1023.792,A -85,B 0,C 180,E1 11007.424,E2 11007.424} C_VEL
LIN {X 0,Y 557.091,Z 983.897,A -85,B 0,C 180,E1 11009.275,E2 11009.275} C_VEL
LIN {X 0,Y 549.989,Z 952.892,A -85,B 0,C 180,E1 11010.877,E2 11010.877} C_VEL
LIN {X 0,Y 537.655,Z 923.03,A -85,B 0,C 180,E1 11012.715,E2 11012.715} C_VEL
LIN {X 0,Y 537.403,Z 923.03,A -85,B 0,C 180,E1 11018.212,E2 11018.212} C_VEL
LIN {X 0,Y 537.313,Z 923.03,A -85,B 0,C 180,E1 11024.672,E2 11024.672} C_VEL
LIN {X 0,Y 537.36,Z 923.03,A -85,B 0,C 180,E1 11029.724,E2 11029.724} C_VEL
LIN {X 0,Y 537.506,Z 923.03,A -85,B 0,C 180,E1 11035.808,E2 11035.808} C_VEL
LIN {X 0,Y 537.569,Z 923.198,A -85,B 0,C 180,E1 11036.538,E2 11036.538} C_VEL
LIN {X 0,Y 551.732,Z 956.301,A -85,B 0,C 180,E1 11038.385,E2 11038.385} C_VEL
LIN {X 0,Y 558.592,Z 982.391,A -85,B 0,C 180,E1 11039.391,E2 11039.391} C_VEL
LIN {X 0,Y 555.933,Z 1022.824,A -85,B 0,C 180,E1 11040.52,E2 11040.52} C_VEL
LIN {X 0,Y 552.916,Z 1035.345,A -85,B 0,C 180,E1 11040.876,E2 11040.876} C_VEL
LIN {X 0,Y 546.506,Z 1053.195,A -85,B 0,C 180,E1 11041.405,E2 11041.405} C_VEL
LIN {X 0,Y 546.228,Z 1055.179,A -85,B 0,C 180,E1 11041.494,E2 11041.494} C_VEL
LIN {X 0,Y 542.399,Z 1094,A -85,B 0,C 180,E1 11043.77,E2 11043.77} C_VEL
LIN {X 0,Y 538.82,Z 1128.178,A -85,B 0,C 180,E1 11046.492,E2 11046.492} C_VEL
LIN {X 0,Y 535.834,Z 1157.562,A -85,B 0,C 180,E1 11049.592,E2 11049.592} C_VEL
LIN {X 0,Y 533.468,Z 1183.017,A -85,B 0,C 180,E1 11053.138,E2 11053.138} C_VEL
LIN {X 0,Y 531.966,Z 1202.916,A -85,B 0,C 180,E1 11056.881,E2 11056.881} C_VEL
LIN {X 0,Y 531.254,Z 1217.033,A -85,B 0,C 180,E1 11060.602,E2 11060.602} C_VEL
LIN {X 0,Y 530.986,Z 1226.212,A -85,B 0,C 180,E1 11064.299,E2 11064.299} C_VEL
LIN {X 0,Y 530.917,Z 1231.065,A -85,B 0,C 180,E1 11068.384,E2 11068.384} C_VEL
LIN {X 0,Y 531.017,Z 1231.126,A -85,B 0,C 180,E1 11071.645,E2 11071.645} C_VEL
LIN {X 0,Y 531.002,Z 1226.474,A -85,B 0,C 180,E1 11075.729,E2 11075.729} C_VEL
LIN {X 0,Y 531.329,Z 1216.294,A -85,B 0,C 180,E1 11079.839,E2 11079.839} C_VEL
LIN {X 0,Y 532.237,Z 1199.953,A -85,B 0,C 180,E1 11083.978,E2 11083.978} C_VEL
LIN {X 0,Y 534.035,Z 1179.069,A -85,B 0,C 180,E1 11087.722,E2 11087.722} C_VEL
LIN {X 0,Y 536.754,Z 1152.377,A -85,B 0,C 180,E1 11091.265,E2 11091.265} C_VEL
LIN {X 0,Y 540.026,Z 1122.254,A -85,B 0,C 180,E1 11094.28,E2 11094.28} C_VEL
LIN {X 0,Y 543.659,Z 1088.733,A -85,B 0,C 180,E1 11096.804,E2 11096.804} C_VEL
LIN {X 0,Y 547.307,Z 1050.383,A -85,B 0,C 180,E1 11098.906,E2 11098.906} C_VEL
LIN {X 0,Y 550.392,Z 1009.335,A -85,B 0,C 180,E1 11100.416,E2 11100.416} C_VEL
LIN {X 0,Y 551.445,Z 980.887,A -85,B 0,C 180,E1 11101.096,E2 11101.096} C_VEL
LIN {X 0,Y 529.7,Z 923.03,A -85,B 0,C 180,E1 11103.33,E2 11103.33} C_VEL
LIN {X 0,Y 529.44,Z 923.03,A -85,B 0,C 180,E1 11109.593,E2 11109.593} C_VEL
LIN {X 0,Y 529.387,Z 923.03,A -85,B 0,C 180,E1 11115.544,E2 11115.544} C_VEL
LIN {X 0,Y 529.452,Z 923.03,A -85,B 0,C 180,E1 11121.107,E2 11121.107} C_VEL
LIN {X 0,Y 529.531,Z 923.03,A -85,B 0,C 180,E1 11127.169,E2 11127.169} C_VEL
LIN {X 0,Y 529.702,Z 923.03,A -85,B 0,C 180,E1 11132.845,E2 11132.845} C_VEL
LIN {X 0,Y 529.839,Z 923.03,A -85,B 0,C 180,E1 11138.239,E2 11138.239} C_VEL
LIN {X 0,Y 529.88,Z 923.03,A -85,B 0,C 180,E1 11143.432,E2 11143.432} C_VEL
LIN {X 0,Y 530.189,Z 923.03,A -85,B 0,C 180,E1 11148.494,E2 11148.494} C_VEL
LIN {X 0,Y 530.43,Z 923.03,A -85,B 0,C 180,E1 11152.257,E2 11152.257} C_VEL
LIN {X 0,Y 538.407,Z 954.816,A -85,B 0,C 180,E1 11153.159,E2 11153.159} C_VEL
LIN {X 0,Y 538.289,Z 994.276,A -85,B 0,C 180,E1 11153.959,E2 11153.959} C_VEL
LIN {X 0,Y 537.551,Z 1022.977,A -85,B 0,C 180,E1 11155.164,E2 11155.164} C_VEL
LIN {X 0,Y 536.369,Z 1048.971,A -85,B 0,C 180,E1 11156.974,E2 11156.974} C_VEL
LIN {X 0,Y 535.09,Z 1070.098,A -85,B 0,C 180,E1 11159.193,E2 11159.193} C_VEL
LIN {X 0,Y 533.883,Z 1086.818,A -85,B 0,C 180,E1 11161.826,E2 11161.826} C_VEL
LIN {X 0,Y 532.932,Z 1097.529,A -85,B 0,C 180,E1 11164.474,E2 11164.474} C_VEL
LIN {X 0,Y 532.499,Z 1102.562,A -85,B 0,C 180,E1 11166.602,E2 11166.602} C_VEL
LIN {X 0,Y 532.131,Z 1104.898,A -85,B 0,C 180,E1 11169.812,E2 11169.812} C_VEL
LIN {X 0,Y 532.182,Z 1102.453,A -85,B 0,C 180,E1 11172.298,E2 11172.298} C_VEL
LIN {X 0,Y 532.581,Z 1094.161,A -85,B 0,C 180,E1 11175.392,E2 11175.392} C_VEL
LIN {X 0,Y 533.208,Z 1079.851,A -85,B 0,C 180,E1 11178.336,E2 11178.336} C_VEL
LIN {X 0,Y 534.195,Z 1060.723,A -85,B 0,C 180,E1 11180.885,E2 11180.885} C_VEL
LIN {X 0,Y 535.141,Z 1036.275,A -85,B 0,C 180,E1 11183.068,E2 11183.068} C_VEL
LIN {X 0,Y 536.129,Z 1009.623,A -85,B 0,C 180,E1 11184.623,E2 11184.623} C_VEL
LIN {X 0,Y 536.631,Z 980.001,A -85,B 0,C 180,E1 11185.635,E2 11185.635} C_VEL
LIN {X 0,Y 536.046,Z 951.194,A -85,B 0,C 180,E1 11186.138,E2 11186.138} C_VEL
LIN {X 0,Y 529.948,Z 923.03,A -85,B 0,C 180,E1 11186.755,E2 11186.755} C_VEL
LIN {X 0,Y 529.508,Z 923.03,A -85,B 0,C 180,E1 11192.837,E2 11192.837} C_VEL
LIN {X 0,Y 529.445,Z 923.03,A -85,B 0,C 180,E1 11198.898,E2 11198.898} C_VEL
LIN {X 0,Y 529.38,Z 923.03,A -85,B 0,C 180,E1 11204.455,E2 11204.455} C_VEL
LIN {X 0,Y 529.465,Z 923.03,A -85,B 0,C 180,E1 11210.409,E2 11210.409} C_VEL
LIN {X 0,Y 529.538,Z 923.03,A -85,B 0,C 180,E1 11215.851,E2 11215.851} C_VEL
LIN {X 0,Y 529.745,Z 923.03,A -85,B 0,C 180,E1 11222.166,E2 11222.166} C_VEL
LIN {X 0,Y 529.894,Z 923.03,A -85,B 0,C 180,E1 11228.227,E2 11228.227} C_VEL
LIN {X 0,Y 530.023,Z 923.03,A -85,B 0,C 180,E1 11233.422,E2 11233.422} C_VEL
LIN {X 0,Y 530.2,Z 923.03,A -85,B 0,C 180,E1 11238.478,E2 11238.478} C_VEL
LIN {X 0,Y 530.472,Z 923.03,A -85,B 0,C 180,E1 11243.443,E2 11243.443} C_VEL
LIN {X 0,Y 530.639,Z 923.03,A -85,B 0,C 180,E1 11248.354,E2 11248.354} C_VEL
LIN {X 0,Y 530.558,Z 923.03,A -85,B 0,C 180,E1 11253.251,E2 11253.251} C_VEL
LIN {X 0,Y 530.397,Z 923.03,A -85,B 0,C 180,E1 11258.174,E2 11258.174} C_VEL
LIN {X 0,Y 530.145,Z 923.03,A -85,B 0,C 180,E1 11264.269,E2 11264.269} C_VEL
LIN {X 0,Y 529.977,Z 923.03,A -85,B 0,C 180,E1 11269.991,E2 11269.991} C_VEL
LIN {X 0,Y 529.799,Z 923.03,A -85,B 0,C 180,E1 11275.312,E2 11275.312} C_VEL
LIN {X 0,Y 529.643,Z 923.03,A -85,B 0,C 180,E1 11281.136,E2 11281.136} C_VEL
LIN {X 0,Y 529.501,Z 923.03,A -85,B 0,C 180,E1 11286.956,E2 11286.956} C_VEL
LIN {X 0,Y 529.535,Z 923.03,A -85,B 0,C 180,E1 11293.201,E2 11293.201} C_VEL
LIN {X 0,Y 529.475,Z 923.03,A -85,B 0,C 180,E1 11298.971,E2 11298.971} C_VEL
LIN {X 0,Y 529.558,Z 923.03,A -85,B 0,C 180,E1 11305.199,E2 11305.199} C_VEL
LIN {X 0,Y 529.61,Z 923.03,A -85,B 0,C 180,E1 11307.52,E2 11307.52} C_VEL
LIN {X 0,Y 545.011,Z 966.796,A -85,B 0,C 180,E1 11309.521,E2 11309.521} C_VEL
LIN {X 0,Y 549.454,Z 984.283,A -85,B 0,C 180,E1 11310.409,E2 11310.409} C_VEL
LIN {X 0,Y 546.118,Z 1023.364,A -85,B 0,C 180,E1 11312.265,E2 11312.265} C_VEL
LIN {X 0,Y 542.389,Z 1059.58,A -85,B 0,C 180,E1 11314.707,E2 11314.707} C_VEL
LIN {X 0,Y 538.885,Z 1090.995,A -85,B 0,C 180,E1 11317.569,E2 11317.569} C_VEL
LIN {X 0,Y 535.803,Z 1118.379,A -85,B 0,C 180,E1 11320.882,E2 11320.882} C_VEL
LIN {X 0,Y 533.648,Z 1140.026,A -85,B 0,C 180,E1 11324.365,E2 11324.365} C_VEL
LIN {X 0,Y 532.116,Z 1157.191,A -85,B 0,C 180,E1 11328.114,E2 11328.114} C_VEL
LIN {X 0,Y 531.371,Z 1169.033,A -85,B 0,C 180,E1 11331.824,E2 11331.824} C_VEL
LIN {X 0,Y 530.986,Z 1176.844,A -85,B 0,C 180,E1 11335.918,E2 11335.918} C_VEL
LIN {X 0,Y 530.805,Z 1179.536,A -85,B 0,C 180,E1 11339.998,E2 11339.998} C_VEL
LIN {X 0,Y 530.937,Z 1177.998,A -85,B 0,C 180,E1 11343.261,E2 11343.261} C_VEL
LIN {X 0,Y 531.393,Z 1171.581,A -85,B 0,C 180,E1 11347.35,E2 11347.35} C_VEL
LIN {X 0,Y 532.152,Z 1159.686,A -85,B 0,C 180,E1 11351.463,E2 11351.463} C_VEL
LIN {X 0,Y 533.679,Z 1142.901,A -85,B 0,C 180,E1 11355.326,E2 11355.326} C_VEL
LIN {X 0,Y 536.099,Z 1120.391,A -85,B 0,C 180,E1 11359.052,E2 11359.052} C_VEL
LIN {X 0,Y 539.138,Z 1094.455,A -85,B 0,C 180,E1 11362.256,E2 11362.256} C_VEL
LIN {X 0,Y 542.714,Z 1063.888,A -85,B 0,C 180,E1 11365.108,E2 11365.108} C_VEL
LIN {X 0,Y 546.575,Z 1027.528,A -85,B 0,C 180,E1 11367.623,E2 11367.623} C_VEL
LIN {X 0,Y 550.028,Z 987.527,A -85,B 0,C 180,E1 11369.57,E2 11369.57} C_VEL
LIN {X 0,Y 549.204,Z 978.013,A -85,B 0,C 180,E1 11370.037,E2 11370.037} C_VEL
LIN {X 0,Y 540.78,Z 948.166,A -85,B 0,C 180,E1 11371.698,E2 11371.698} C_VEL
LIN {X 0,Y 529.721,Z 923.03,A -85,B 0,C 180,E1 11373.374,E2 11373.374} C_VEL
LIN {X 0,Y 529.397,Z 923.03,A -85,B 0,C 180,E1 11379.614,E2 11379.614} C_VEL
LIN {X 0,Y 529.419,Z 923.03,A -85,B 0,C 180,E1 11385.523,E2 11385.523} C_VEL
LIN {X 0,Y 529.45,Z 923.03,A -85,B 0,C 180,E1 11391.128,E2 11391.128} C_VEL
LIN {X 0,Y 529.622,Z 923.03,A -85,B 0,C 180,E1 11395.768,E2 11395.768} C_VEL
LIN {X 0,Y 543.842,Z 954.978,A -85,B 0,C 180,E1 11397.786,E2 11397.786} C_VEL
LIN {X 0,Y 551.852,Z 982.424,A -85,B 0,C 180,E1 11398.968,E2 11398.968} C_VEL
LIN {X 0,Y 548.768,Z 1025.459,A -85,B 0,C 180,E1 11400.222,E2 11400.222} C_VEL
LIN {X 0,Y 546.228,Z 1055.179,A -85,B 0,C 180,E1 11401.494,E2 11401.494} C_VEL
LIN {X 0,Y 541.082,Z 1070.827,A -85,B 0,C 180,E1 11402.134,E2 11402.134} C_VEL
LIN {X 0,Y 536,Z 1085.963,A -85,B 0,C 180,E1 11402.889,E2 11402.889} C_VEL
LIN {X 0,Y 532.163,Z 1120.977,A -85,B 0,C 180,E1 11405.55,E2 11405.55} C_VEL
LIN {X 0,Y 528.605,Z 1153.525,A -85,B 0,C 180,E1 11408.862,E2 11408.862} C_VEL
LIN {X 0,Y 525.997,Z 1179.879,A -85,B 0,C 180,E1 11412.46,E2 11412.46} C_VEL
LIN {X 0,Y 524.305,Z 1200.548,A -85,B 0,C 180,E1 11416.261,E2 11416.261} C_VEL
LIN {X 0,Y 523.38,Z 1216.592,A -85,B 0,C 180,E1 11420.46,E2 11420.46} C_VEL
LIN {X 0,Y 523.092,Z 1225.803,A -85,B 0,C 180,E1 11424.212,E2 11424.212} C_VEL
LIN {X 0,Y 523.023,Z 1230.674,A -85,B 0,C 180,E1 11428.359,E2 11428.359} C_VEL
LIN {X 0,Y 523.121,Z 1230.721,A -85,B 0,C 180,E1 11431.67,E2 11431.67} C_VEL
LIN {X 0,Y 523.109,Z 1226.024,A -85,B 0,C 180,E1 11435.817,E2 11435.817} C_VEL
LIN {X 0,Y 523.443,Z 1215.77,A -85,B 0,C 180,E1 11439.988,E2 11439.988} C_VEL
LIN {X 0,Y 524.362,Z 1200.324,A -85,B 0,C 180,E1 11443.98,E2 11443.98} C_VEL
LIN {X 0,Y 526.291,Z 1178.253,A -85,B 0,C 180,E1 11447.992,E2 11447.992} C_VEL
LIN {X 0,Y 528.962,Z 1153.21,A -85,B 0,C 180,E1 11451.374,E2 11451.374} C_VEL
LIN {X 0,Y 532.427,Z 1122.408,A -85,B 0,C 180,E1 11454.516,E2 11454.516} C_VEL
LIN {X 0,Y 536.322,Z 1087.881,A -85,B 0,C 180,E1 11457.145,E2 11457.145} C_VEL
LIN {X 0,Y 540.076,Z 1049.376,A -85,B 0,C 180,E1 11459.273,E2 11459.273} C_VEL
LIN {X 0,Y 543.352,Z 1006.868,A -85,B 0,C 180,E1 11460.827,E2 11460.827} C_VEL
LIN {X 0,Y 544.209,Z 982.583,A -85,B 0,C 180,E1 11461.427,E2 11461.427} C_VEL
LIN {X 0,Y 521.763,Z 923.03,A -85,B 0,C 180,E1 11463.773,E2 11463.773} C_VEL
LIN {X 0,Y 521.566,Z 923.03,A -85,B 0,C 180,E1 11469.612,E2 11469.612} C_VEL
LIN {X 0,Y 521.495,Z 923.03,A -85,B 0,C 180,E1 11475.941,E2 11475.941} C_VEL
LIN {X 0,Y 521.545,Z 923.03,A -85,B 0,C 180,E1 11481.487,E2 11481.487} C_VEL
LIN {X 0,Y 521.656,Z 923.03,A -85,B 0,C 180,E1 11487.164,E2 11487.164} C_VEL
LIN {X 0,Y 521.788,Z 923.03,A -85,B 0,C 180,E1 11492.398,E2 11492.398} C_VEL
LIN {X 0,Y 521.917,Z 923.03,A -85,B 0,C 180,E1 11497.92,E2 11497.92} C_VEL
LIN {X 0,Y 521.944,Z 923.03,A -85,B 0,C 180,E1 11503.173,E2 11503.173} C_VEL
LIN {X 0,Y 522.255,Z 923.03,A -85,B 0,C 180,E1 11508.316,E2 11508.316} C_VEL
LIN {X 0,Y 522.49,Z 923.03,A -85,B 0,C 180,E1 11511.901,E2 11511.901} C_VEL
LIN {X 0,Y 531.082,Z 956.375,A -85,B 0,C 180,E1 11512.887,E2 11512.887} C_VEL
LIN {X 0,Y 530.892,Z 994.646,A -85,B 0,C 180,E1 11513.669,E2 11513.669} C_VEL
LIN {X 0,Y 530.079,Z 1023.529,A -85,B 0,C 180,E1 11514.891,E2 11514.891} C_VEL
LIN {X 0,Y 528.824,Z 1049.693,A -85,B 0,C 180,E1 11516.726,E2 11516.726} C_VEL
LIN {X 0,Y 527.49,Z 1070.952,A -85,B 0,C 180,E1 11518.976,E2 11518.976} C_VEL
LIN {X 0,Y 526.182,Z 1087.73,A -85,B 0,C 180,E1 11521.647,E2 11521.647} C_VEL
LIN {X 0,Y 525.122,Z 1099.085,A -85,B 0,C 180,E1 11524.541,E2 11524.541} C_VEL
LIN {X 0,Y 524.669,Z 1103.728,A -85,B 0,C 180,E1 11526.617,E2 11526.617} C_VEL
LIN {X 0,Y 524.398,Z 1105.588,A -85,B 0,C 180,E1 11528.286,E2 11528.286} C_VEL
LIN {X 0,Y 524.343,Z 1104.564,A -85,B 0,C 180,E1 11531.477,E2 11531.477} C_VEL
LIN {X 0,Y 524.612,Z 1097.844,A -85,B 0,C 180,E1 11534.6,E2 11534.6} C_VEL
LIN {X 0,Y 525.125,Z 1085.672,A -85,B 0,C 180,E1 11537.527,E2 11537.527} C_VEL
LIN {X 0,Y 526.031,Z 1067.447,A -85,B 0,C 180,E1 11540.298,E2 11540.298} C_VEL
LIN {X 0,Y 527.099,Z 1044.466,A -85,B 0,C 180,E1 11542.62,E2 11542.62} C_VEL
LIN {X 0,Y 528.214,Z 1017.971,A -85,B 0,C 180,E1 11544.397,E2 11544.397} C_VEL
LIN {X 0,Y 528.842,Z 987.999,A -85,B 0,C 180,E1 11545.609,E2 11545.609} C_VEL
LIN {X 0,Y 528.423,Z 952.61,A -85,B 0,C 180,E1 11546.302,E2 11546.302} C_VEL
LIN {X 0,Y 521.979,Z 923.03,A -85,B 0,C 180,E1 11547.003,E2 11547.003} C_VEL
LIN {X 0,Y 521.592,Z 923.03,A -85,B 0,C 180,E1 11553.4,E2 11553.4} C_VEL
LIN {X 0,Y 521.562,Z 923.03,A -85,B 0,C 180,E1 11559.6,E2 11559.6} C_VEL
LIN {X 0,Y 521.496,Z 923.03,A -85,B 0,C 180,E1 11565.923,E2 11565.923} C_VEL
LIN {X 0,Y 521.554,Z 923.03,A -85,B 0,C 180,E1 11571.472,E2 11571.472} C_VEL
LIN {X 0,Y 521.644,Z 923.03,A -85,B 0,C 180,E1 11577.151,E2 11577.151} C_VEL
LIN {X 0,Y 521.876,Z 923.03,A -85,B 0,C 180,E1 11582.387,E2 11582.387} C_VEL
LIN {X 0,Y 521.956,Z 923.03,A -85,B 0,C 180,E1 11587.888,E2 11587.888} C_VEL
LIN {X 0,Y 522.09,Z 923.03,A -85,B 0,C 180,E1 11593.162,E2 11593.162} C_VEL
LIN {X 0,Y 522.329,Z 923.03,A -85,B 0,C 180,E1 11599.625,E2 11599.625} C_VEL
LIN {X 0,Y 522.654,Z 923.03,A -85,B 0,C 180,E1 11605.01,E2 11605.01} C_VEL
LIN {X 0,Y 522.918,Z 923.03,A -85,B 0,C 180,E1 11609.985,E2 11609.985} C_VEL
LIN {X 0,Y 522.582,Z 923.03,A -85,B 0,C 180,E1 11616.627,E2 11616.627} C_VEL
LIN {X 0,Y 522.336,Z 923.03,A -85,B 0,C 180,E1 11621.668,E2 11621.668} C_VEL
LIN {X 0,Y 522.135,Z 923.03,A -85,B 0,C 180,E1 11627.239,E2 11627.239} C_VEL
LIN {X 0,Y 521.96,Z 923.03,A -85,B 0,C 180,E1 11632.113,E2 11632.113} C_VEL
LIN {X 0,Y 521.854,Z 923.03,A -85,B 0,C 180,E1 11637.581,E2 11637.581} C_VEL
LIN {X 0,Y 521.695,Z 923.03,A -85,B 0,C 180,E1 11643.369,E2 11643.369} C_VEL
LIN {X 0,Y 521.594,Z 923.03,A -85,B 0,C 180,E1 11649.572,E2 11649.572} C_VEL
LIN {X 0,Y 521.628,Z 923.03,A -85,B 0,C 180,E1 11655.95,E2 11655.95} C_VEL
LIN {X 0,Y 521.517,Z 923.03,A -85,B 0,C 180,E1 11661.444,E2 11661.444} C_VEL
LIN {X 0,Y 521.656,Z 923.03,A -85,B 0,C 180,E1 11667.11,E2 11667.11} C_VEL
LIN {X 0,Y 536.575,Z 965.058,A -85,B 0,C 180,E1 11669.032,E2 11669.032} C_VEL
LIN {X 0,Y 542.18,Z 985.489,A -85,B 0,C 180,E1 11670.104,E2 11670.104} C_VEL
LIN {X 0,Y 538.681,Z 1024.787,A -85,B 0,C 180,E1 11672.016,E2 11672.016} C_VEL
LIN {X 0,Y 534.887,Z 1060.486,A -85,B 0,C 180,E1 11674.468,E2 11674.468} C_VEL
LIN {X 0,Y 531.267,Z 1091.898,A -85,B 0,C 180,E1 11677.377,E2 11677.377} C_VEL
LIN {X 0,Y 528.089,Z 1119.107,A -85,B 0,C 180,E1 11680.724,E2 11680.724} C_VEL
LIN {X 0,Y 525.795,Z 1141.17,A -85,B 0,C 180,E1 11684.347,E2 11684.347} C_VEL
LIN {X 0,Y 524.18,Z 1159.319,A -85,B 0,C 180,E1 11688.465,E2 11688.465} C_VEL
LIN {X 0,Y 523.388,Z 1171.271,A -85,B 0,C 180,E1 11692.533,E2 11692.533} C_VEL
LIN {X 0,Y 523.026,Z 1178.094,A -85,B 0,C 180,E1 11696.686,E2 11696.686} C_VEL
LIN {X 0,Y 522.915,Z 1179.933,A -85,B 0,C 180,E1 11699.998,E2 11699.998} C_VEL
LIN {X 0,Y 523.061,Z 1178.428,A -85,B 0,C 180,E1 11703.311,E2 11703.311} C_VEL
LIN {X 0,Y 523.531,Z 1172.03,A -85,B 0,C 180,E1 11707.461,E2 11707.461} C_VEL
LIN {X 0,Y 524.368,Z 1160.144,A -85,B 0,C 180,E1 11711.636,E2 11711.636} C_VEL
LIN {X 0,Y 526.075,Z 1142.62,A -85,B 0,C 180,E1 11715.699,E2 11715.699} C_VEL
LIN {X 0,Y 528.711,Z 1119.923,A -85,B 0,C 180,E1 11719.468,E2 11719.468} C_VEL
LIN {X 0,Y 532.031,Z 1093.087,A -85,B 0,C 180,E1 11722.783,E2 11722.783} C_VEL
LIN {X 0,Y 536.12,Z 1059.91,A -85,B 0,C 180,E1 11725.839,E2 11725.839} C_VEL
LIN {X 0,Y 540.121,Z 1022.995,A -85,B 0,C 180,E1 11728.312,E2 11728.312} C_VEL
LIN {X 0,Y 543.423,Z 985.034,A -85,B 0,C 180,E1 11730.125,E2 11730.125} C_VEL
LIN {X 0,Y 535.322,Z 953.354,A -85,B 0,C 180,E1 11731.976,E2 11731.976} C_VEL
LIN {X 0,Y 523.824,Z 928.343,A -85,B 0,C 180,E1 11733.77,E2 11733.77} C_VEL
LIN {X 0,Y 521.783,Z 923.03,A -85,B 0,C 180,E1 11734.143,E2 11734.143} C_VEL
LIN {X 0,Y 521.519,Z 923.03,A -85,B 0,C 180,E1 11739.599,E2 11739.599} C_VEL
LIN {X 0,Y 521.491,Z 923.03,A -85,B 0,C 180,E1 11745.964,E2 11745.964} C_VEL
LIN {X 0,Y 521.54,Z 923.03,A -85,B 0,C 180,E1 11751.468,E2 11751.468} C_VEL
LIN {X 0,Y 521.674,Z 923.03,A -85,B 0,C 180,E1 11754.967,E2 11754.967} C_VEL
LIN {X 0,Y 526.576,Z 933.555,A -85,B 0,C 180,E1 11755.783,E2 11755.783} C_VEL
LIN {X 0,Y 538.254,Z 959.672,A -85,B 0,C 180,E1 11757.457,E2 11757.457} C_VEL
LIN {X 0,Y 545.062,Z 984.287,A -85,B 0,C 180,E1 11758.566,E2 11758.566} C_VEL
LIN {X 0,Y 541.74,Z 1027.3,A -85,B 0,C 180,E1 11759.882,E2 11759.882} C_VEL
LIN {X 0,Y 537.736,Z 1068.66,A -85,B 0,C 180,E1 11761.828,E2 11761.828} C_VEL
LIN {X 0,Y 536,Z 1085.963,A -85,B 0,C 180,E1 11762.889,E2 11762.889} C_VEL
LIN {X 0,Y 530.791,Z 1100.73,A -85,B 0,C 180,E1 11763.738,E2 11763.738} C_VEL
LIN {X 0,Y 525.45,Z 1114.863,A -85,B 0,C 180,E1 11764.699,E2 11764.699} C_VEL
LIN {X 0,Y 521.92,Z 1145.513,A -85,B 0,C 180,E1 11767.684,E2 11767.684} C_VEL
LIN {X 0,Y 518.971,Z 1172.344,A -85,B 0,C 180,E1 11771.117,E2 11771.117} C_VEL
LIN {X 0,Y 516.859,Z 1194.941,A -85,B 0,C 180,E1 11774.978,E2 11774.978} C_VEL
LIN {X 0,Y 515.752,Z 1211.327,A -85,B 0,C 180,E1 11778.837,E2 11778.837} C_VEL
LIN {X 0,Y 515.323,Z 1221.865,A -85,B 0,C 180,E1 11782.433,E2 11782.433} C_VEL
LIN {X 0,Y 515.174,Z 1228.941,A -85,B 0,C 180,E1 11786.652,E2 11786.652} C_VEL
LIN {X 0,Y 515.161,Z 1230.739,A -85,B 0,C 180,E1 11790.015,E2 11790.015} C_VEL
LIN {X 0,Y 515.189,Z 1228.076,A -85,B 0,C 180,E1 11794.274,E2 11794.274} C_VEL
LIN {X 0,Y 515.41,Z 1220.089,A -85,B 0,C 180,E1 11798.444,E2 11798.444} C_VEL
LIN {X 0,Y 516.125,Z 1206.128,A -85,B 0,C 180,E1 11802.698,E2 11802.698} C_VEL
LIN {X 0,Y 517.674,Z 1186.631,A -85,B 0,C 180,E1 11806.745,E2 11806.745} C_VEL
LIN {X 0,Y 520.17,Z 1162.469,A -85,B 0,C 180,E1 11810.415,E2 11810.415} C_VEL
LIN {X 0,Y 523.564,Z 1133.39,A -85,B 0,C 180,E1 11813.733,E2 11813.733} C_VEL
LIN {X 0,Y 527.534,Z 1099.864,A -85,B 0,C 180,E1 11816.601,E2 11816.601} C_VEL
LIN {X 0,Y 531.406,Z 1062.979,A -85,B 0,C 180,E1 11818.922,E2 11818.922} C_VEL
LIN {X 0,Y 535.146,Z 1022.301,A -85,B 0,C 180,E1 11820.689,E2 11820.689} C_VEL
LIN {X 0,Y 537.02,Z 984.588,A -85,B 0,C 180,E1 11821.744,E2 11821.744} C_VEL
LIN {X 0,Y 513.818,Z 923.03,A -85,B 0,C 180,E1 11824.239,E2 11824.239} C_VEL
LIN {X 0,Y 513.605,Z 923.03,A -85,B 0,C 180,E1 11830.351,E2 11830.351} C_VEL
LIN {X 0,Y 513.526,Z 923.03,A -85,B 0,C 180,E1 11835.074,E2 11835.074} C_VEL
LIN {X 0,Y 513.624,Z 923.03,A -85,B 0,C 180,E1 11839.917,E2 11839.917} C_VEL
LIN {X 0,Y 513.632,Z 923.03,A -85,B 0,C 180,E1 11846.017,E2 11846.017} C_VEL
LIN {X 0,Y 513.809,Z 923.03,A -85,B 0,C 180,E1 11851.942,E2 11851.942} C_VEL
LIN {X 0,Y 513.963,Z 923.03,A -85,B 0,C 180,E1 11857.531,E2 11857.531} C_VEL
LIN {X 0,Y 514.021,Z 923.03,A -85,B 0,C 180,E1 11862.906,E2 11862.906} C_VEL
LIN {X 0,Y 514.319,Z 923.03,A -85,B 0,C 180,E1 11868.133,E2 11868.133} C_VEL
LIN {X 0,Y 514.556,Z 923.03,A -85,B 0,C 180,E1 11871.505,E2 11871.505} C_VEL
LIN {X 0,Y 523.64,Z 957.083,A -85,B 0,C 180,E1 11872.582,E2 11872.582} C_VEL
LIN {X 0,Y 523.425,Z 996.724,A -85,B 0,C 180,E1 11873.423,E2 11873.423} C_VEL
LIN {X 0,Y 522.594,Z 1026.024,A -85,B 0,C 180,E1 11874.713,E2 11874.713} C_VEL
LIN {X 0,Y 521.263,Z 1051.654,A -85,B 0,C 180,E1 11876.574,E2 11876.574} C_VEL
LIN {X 0,Y 519.773,Z 1073.344,A -85,B 0,C 180,E1 11878.961,E2 11878.961} C_VEL
LIN {X 0,Y 518.409,Z 1089.702,A -85,B 0,C 180,E1 11881.672,E2 11881.672} C_VEL
LIN {X 0,Y 517.305,Z 1100.645,A -85,B 0,C 180,E1 11884.609,E2 11884.609} C_VEL
LIN {X 0,Y 516.829,Z 1105.032,A -85,B 0,C 180,E1 11886.718,E2 11886.718} C_VEL
LIN {X 0,Y 516.568,Z 1106.646,A -85,B 0,C 180,E1 11888.412,E2 11888.412} C_VEL
LIN {X 0,Y 516.452,Z 1106.66,A -85,B 0,C 180,E1 11890.113,E2 11890.113} C_VEL
LIN {X 0,Y 516.539,Z 1103.608,A -85,B 0,C 180,E1 11892.676,E2 11892.676} C_VEL
LIN {X 0,Y 516.938,Z 1095.036,A -85,B 0,C 180,E1 11895.69,E2 11895.69} C_VEL
LIN {X 0,Y 517.59,Z 1081.506,A -85,B 0,C 180,E1 11898.483,E2 11898.483} C_VEL
LIN {X 0,Y 518.553,Z 1062.754,A -85,B 0,C 180,E1 11901.049,E2 11901.049} C_VEL
LIN {X 0,Y 519.561,Z 1039.37,A -85,B 0,C 180,E1 11903.216,E2 11903.216} C_VEL
LIN {X 0,Y 520.664,Z 1012.006,A -85,B 0,C 180,E1 11904.889,E2 11904.889} C_VEL
LIN {X 0,Y 521.196,Z 982.503,A -85,B 0,C 180,E1 11905.944,E2 11905.944} C_VEL
LIN {X 0,Y 520.539,Z 952.964,A -85,B 0,C 180,E1 11906.491,E2 11906.491} C_VEL
LIN {X 0,Y 514.033,Z 923.03,A -85,B 0,C 180,E1 11907.23,E2 11907.23} C_VEL
LIN {X 0,Y 513.612,Z 923.03,A -85,B 0,C 180,E1 11913.989,E2 11913.989} C_VEL
LIN {X 0,Y 513.628,Z 923.03,A -85,B 0,C 180,E1 11920.083,E2 11920.083} C_VEL
LIN {X 0,Y 513.526,Z 923.03,A -85,B 0,C 180,E1 11925.056,E2 11925.056} C_VEL
LIN {X 0,Y 513.652,Z 923.03,A -85,B 0,C 180,E1 11929.9,E2 11929.9} C_VEL
LIN {X 0,Y 513.616,Z 923.03,A -85,B 0,C 180,E1 11935.999,E2 11935.999} C_VEL
LIN {X 0,Y 513.89,Z 923.03,A -85,B 0,C 180,E1 11941.92,E2 11941.92} C_VEL
LIN {X 0,Y 514.001,Z 923.03,A -85,B 0,C 180,E1 11947.517,E2 11947.517} C_VEL
LIN {X 0,Y 514.203,Z 923.03,A -85,B 0,C 180,E1 11952.896,E2 11952.896} C_VEL
LIN {X 0,Y 514.363,Z 923.03,A -85,B 0,C 180,E1 11958.119,E2 11958.119} C_VEL
LIN {X 0,Y 514.651,Z 923.03,A -85,B 0,C 180,E1 11963.241,E2 11963.241} C_VEL
LIN {X 0,Y 514.853,Z 923.03,A -85,B 0,C 180,E1 11968.303,E2 11968.303} C_VEL
LIN {X 0,Y 514.748,Z 923.03,A -85,B 0,C 180,E1 11973.497,E2 11973.497} C_VEL
LIN {X 0,Y 514.585,Z 923.03,A -85,B 0,C 180,E1 11978.427,E2 11978.427} C_VEL
LIN {X 0,Y 514.318,Z 923.03,A -85,B 0,C 180,E1 11984.166,E2 11984.166} C_VEL
LIN {X 0,Y 514.131,Z 923.03,A -85,B 0,C 180,E1 11989.855,E2 11989.855} C_VEL
LIN {X 0,Y 513.952,Z 923.03,A -85,B 0,C 180,E1 11996.15,E2 11996.15} C_VEL
LIN {X 0,Y 513.799,Z 923.03,A -85,B 0,C 180,E1 12001.943,E2 12001.943} C_VEL
LIN {X 0,Y 513.651,Z 923.03,A -85,B 0,C 180,E1 12008.132,E2 12008.132} C_VEL
LIN {X 0,Y 513.661,Z 923.03,A -85,B 0,C 180,E1 12014.887,E2 12014.887} C_VEL
LIN {X 0,Y 513.638,Z 923.03,A -85,B 0,C 180,E1 12019.869,E2 12019.869} C_VEL
LIN {X 0,Y 513.764,Z 923.03,A -85,B 0,C 180,E1 12026.631,E2 12026.631} C_VEL
LIN {X 0,Y 529.768,Z 968.424,A -85,B 0,C 180,E1 12028.802,E2 12028.802} C_VEL
LIN {X 0,Y 534.807,Z 987.918,A -85,B 0,C 180,E1 12029.85,E2 12029.85} C_VEL
LIN {X 0,Y 531.23,Z 1026.596,A -85,B 0,C 180,E1 12031.787,E2 12031.787} C_VEL
LIN {X 0,Y 527.369,Z 1061.421,A -85,B 0,C 180,E1 12034.226,E2 12034.226} C_VEL
LIN {X 0,Y 523.727,Z 1091.977,A -85,B 0,C 180,E1 12037.095,E2 12037.095} C_VEL
LIN {X 0,Y 520.436,Z 1118.882,A -85,B 0,C 180,E1 12040.429,E2 12040.429} C_VEL
LIN {X 0,Y 518.002,Z 1141.742,A -85,B 0,C 180,E1 12044.221,E2 12044.221} C_VEL
LIN {X 0,Y 516.366,Z 1159.049,A -85,B 0,C 180,E1 12048.178,E2 12048.178} C_VEL
LIN {X 0,Y 515.514,Z 1171.526,A -85,B 0,C 180,E1 12052.418,E2 12052.418} C_VEL
LIN {X 0,Y 515.14,Z 1178.438,A -85,B 0,C 180,E1 12056.635,E2 12056.635} C_VEL
LIN {X 0,Y 515.026,Z 1180.329,A -85,B 0,C 180,E1 12059.998,E2 12059.998} C_VEL
LIN {X 0,Y 515.176,Z 1178.866,A -85,B 0,C 180,E1 12063.361,E2 12063.361} C_VEL
LIN {X 0,Y 515.69,Z 1172.495,A -85,B 0,C 180,E1 12067.575,E2 12067.575} C_VEL
LIN {X 0,Y 516.601,Z 1160.63,A -85,B 0,C 180,E1 12071.813,E2 12071.813} C_VEL
LIN {X 0,Y 518.405,Z 1143.138,A -85,B 0,C 180,E1 12075.936,E2 12075.936} C_VEL
LIN {X 0,Y 521.203,Z 1120.459,A -85,B 0,C 180,E1 12079.76,E2 12079.76} C_VEL
LIN {X 0,Y 524.763,Z 1093.285,A -85,B 0,C 180,E1 12083.162,E2 12083.162} C_VEL
LIN {X 0,Y 529.023,Z 1060.781,A -85,B 0,C 180,E1 12086.197,E2 12086.197} C_VEL
LIN {X 0,Y 533.238,Z 1023.799,A -85,B 0,C 180,E1 12088.72,E2 12088.72} C_VEL
LIN {X 0,Y 536.382,Z 985.819,A -85,B 0,C 180,E1 12090.599,E2 12090.599} C_VEL
LIN {X 0,Y 528.93,Z 956.069,A -85,B 0,C 180,E1 12092.429,E2 12092.429} C_VEL
LIN {X 0,Y 518.202,Z 932.614,A -85,B 0,C 180,E1 12094.236,E2 12094.236} C_VEL
LIN {X 0,Y 513.767,Z 923.03,A -85,B 0,C 180,E1 12095.103,E2 12095.103} C_VEL
LIN {X 0,Y 513.576,Z 923.03,A -85,B 0,C 180,E1 12100.337,E2 12100.337} C_VEL
LIN {X 0,Y 513.518,Z 923.03,A -85,B 0,C 180,E1 12105.097,E2 12105.097} C_VEL
LIN {X 0,Y 513.647,Z 923.03,A -85,B 0,C 180,E1 12111.867,E2 12111.867} C_VEL
LIN {X 0,Y 513.716,Z 923.487,A -85,B 0,C 180,E1 12114.062,E2 12114.062} C_VEL
LIN {X 0,Y 516.314,Z 928.885,A -85,B 0,C 180,E1 12114.551,E2 12114.551} C_VEL
LIN {X 0,Y 528.447,Z 953.43,A -85,B 0,C 180,E1 12116.48,E2 12116.48} C_VEL
LIN {X 0,Y 537.11,Z 979.864,A -85,B 0,C 180,E1 12117.87,E2 12117.87} C_VEL
LIN {X 0,Y 538.212,Z 988.325,A -85,B 0,C 180,E1 12118.197,E2 12118.197} C_VEL
LIN {X 0,Y 534.476,Z 1032.149,A -85,B 0,C 180,E1 12119.652,E2 12119.652} C_VEL
LIN {X 0,Y 530.157,Z 1072.992,A -85,B 0,C 180,E1 12121.699,E2 12121.699} C_VEL
LIN {X 0,Y 526.063,Z 1109.675,A -85,B 0,C 180,E1 12124.268,E2 12124.268} C_VEL
LIN {X 0,Y 525.45,Z 1114.863,A -85,B 0,C 180,E1 12124.699,E2 12124.699} C_VEL
LIN {X 0,Y 520.102,Z 1128.491,A -85,B 0,C 180,E1 12125.769,E2 12125.769} C_VEL
LIN {X 0,Y 514.873,Z 1141.401,A -85,B 0,C 180,E1 12126.934,E2 12126.934} C_VEL
LIN {X 0,Y 511.514,Z 1170.441,A -85,B 0,C 180,E1 12130.607,E2 12130.607} C_VEL
LIN {X 0,Y 509.173,Z 1193.435,A -85,B 0,C 180,E1 12134.525,E2 12134.525} C_VEL
LIN {X 0,Y 507.905,Z 1210.799,A -85,B 0,C 180,E1 12138.63,E2 12138.63} C_VEL
LIN {X 0,Y 507.462,Z 1221.469,A -85,B 0,C 180,E1 12142.315,E2 12142.315} C_VEL
LIN {X 0,Y 507.283,Z 1228.557,A -85,B 0,C 180,E1 12146.6,E2 12146.6} C_VEL
LIN {X 0,Y 507.284,Z 1230.333,A -85,B 0,C 180,E1 12150.015,E2 12150.015} C_VEL
LIN {X 0,Y 507.295,Z 1227.627,A -85,B 0,C 180,E1 12154.341,E2 12154.341} C_VEL
LIN {X 0,Y 507.521,Z 1219.577,A -85,B 0,C 180,E1 12158.576,E2 12158.576} C_VEL
LIN {X 0,Y 508.278,Z 1205.475,A -85,B 0,C 180,E1 12162.898,E2 12162.898} C_VEL
LIN {X 0,Y 509.947,Z 1185.688,A -85,B 0,C 180,E1 12167.029,E2 12167.029} C_VEL
LIN {X 0,Y 512.538,Z 1161.466,A -85,B 0,C 180,E1 12170.733,E2 12170.733} C_VEL
LIN {X 0,Y 516.053,Z 1132.107,A -85,B 0,C 180,E1 12174.1,E2 12174.1} C_VEL
LIN {X 0,Y 520.067,Z 1099.655,A -85,B 0,C 180,E1 12176.897,E2 12176.897} C_VEL
LIN {X 0,Y 523.987,Z 1063.508,A -85,B 0,C 180,E1 12179.21,E2 12179.21} C_VEL
LIN {X 0,Y 527.756,Z 1024.108,A -85,B 0,C 180,E1 12180.969,E2 12180.969} C_VEL
LIN {X 0,Y 529.703,Z 986.014,A -85,B 0,C 180,E1 12182.084,E2 12182.084} C_VEL
LIN {X 0,Y 505.897,Z 923.03,A -85,B 0,C 180,E1 12184.658,E2 12184.658} C_VEL
LIN {X 0,Y 505.6,Z 923.03,A -85,B 0,C 180,E1 12191.126,E2 12191.126} C_VEL
LIN {X 0,Y 505.581,Z 923.03,A -85,B 0,C 180,E1 12196.575,E2 12196.575} C_VEL
LIN {X 0,Y 505.711,Z 923.03,A -85,B 0,C 180,E1 12203.303,E2 12203.303} C_VEL
LIN {X 0,Y 505.826,Z 923.03,A -85,B 0,C 180,E1 12210.057,E2 12210.057} C_VEL
LIN {X 0,Y 505.972,Z 923.03,A -85,B 0,C 180,E1 12215.287,E2 12215.287} C_VEL
LIN {X 0,Y 506.093,Z 923.03,A -85,B 0,C 180,E1 12220.828,E2 12220.828} C_VEL
LIN {X 0,Y 506.271,Z 923.03,A -85,B 0,C 180,E1 12226.187,E2 12226.187} C_VEL
LIN {X 0,Y 506.602,Z 923.03,A -85,B 0,C 180,E1 12231.096,E2 12231.096} C_VEL
LIN {X 0,Y 516.321,Z 958.167,A -85,B 0,C 180,E1 12232.271,E2 12232.271} C_VEL
LIN {X 0,Y 516.021,Z 998.589,A -85,B 0,C 180,E1 12233.163,E2 12233.163} C_VEL
LIN {X 0,Y 515.096,Z 1028.525,A -85,B 0,C 180,E1 12234.531,E2 12234.531} C_VEL
LIN {X 0,Y 513.712,Z 1053.696,A -85,B 0,C 180,E1 12236.418,E2 12236.418} C_VEL
LIN {X 0,Y 512.19,Z 1074.266,A -85,B 0,C 180,E1 12238.734,E2 12238.734} C_VEL
LIN {X 0,Y 510.741,Z 1090.63,A -85,B 0,C 180,E1 12241.485,E2 12241.485} C_VEL
LIN {X 0,Y 509.631,Z 1101.023,A -85,B 0,C 180,E1 12244.253,E2 12244.253} C_VEL
LIN {X 0,Y 508.978,Z 1106.285,A -85,B 0,C 180,E1 12246.822,E2 12246.822} C_VEL
LIN {X 0,Y 508.722,Z 1107.715,A -85,B 0,C 180,E1 12248.543,E2 12248.543} C_VEL
LIN {X 0,Y 508.619,Z 1106.605,A -85,B 0,C 180,E1 12251.306,E2 12251.306} C_VEL
LIN {X 0,Y 508.928,Z 1099.993,A -85,B 0,C 180,E1 12254.52,E2 12254.52} C_VEL
LIN {X 0,Y 509.453,Z 1087.939,A -85,B 0,C 180,E1 12257.546,E2 12257.546} C_VEL
LIN {X 0,Y 510.374,Z 1070.12,A -85,B 0,C 180,E1 12260.36,E2 12260.36} C_VEL
LIN {X 0,Y 511.492,Z 1047.661,A -85,B 0,C 180,E1 12262.741,E2 12262.741} C_VEL
LIN {X 0,Y 512.668,Z 1021.201,A -85,B 0,C 180,E1 12264.605,E2 12264.605} C_VEL
LIN {X 0,Y 513.373,Z 992.649,A -85,B 0,C 180,E1 12265.851,E2 12265.851} C_VEL
LIN {X 0,Y 513.121,Z 955.364,A -85,B 0,C 180,E1 12266.639,E2 12266.639} C_VEL
LIN {X 0,Y 506.122,Z 923.03,A -85,B 0,C 180,E1 12267.405,E2 12267.405} C_VEL
LIN {X 0,Y 505.664,Z 923.03,A -85,B 0,C 180,E1 12273.184,E2 12273.184} C_VEL
LIN {X 0,Y 505.661,Z 923.03,A -85,B 0,C 180,E1 12278.998,E2 12278.998} C_VEL
LIN {X 0,Y 505.554,Z 923.03,A -85,B 0,C 180,E1 12284.147,E2 12284.147} C_VEL
LIN {X 0,Y 505.625,Z 923.03,A -85,B 0,C 180,E1 12288.876,E2 12288.876} C_VEL
LIN {X 0,Y 505.703,Z 923.03,A -85,B 0,C 180,E1 12295.393,E2 12295.393} C_VEL
LIN {X 0,Y 505.925,Z 923.03,A -85,B 0,C 180,E1 12301.438,E2 12301.438} C_VEL
LIN {X 0,Y 506.096,Z 923.03,A -85,B 0,C 180,E1 12307.763,E2 12307.763} C_VEL
LIN {X 0,Y 506.283,Z 923.03,A -85,B 0,C 180,E1 12312.772,E2 12312.772} C_VEL
LIN {X 0,Y 506.447,Z 923.03,A -85,B 0,C 180,E1 12317.93,E2 12317.93} C_VEL
LIN {X 0,Y 506.733,Z 923.03,A -85,B 0,C 180,E1 12323.135,E2 12323.135} C_VEL
LIN {X 0,Y 506.95,Z 923.03,A -85,B 0,C 180,E1 12328.277,E2 12328.277} C_VEL
LIN {X 0,Y 506.887,Z 923.03,A -85,B 0,C 180,E1 12333.403,E2 12333.403} C_VEL
LIN {X 0,Y 506.662,Z 923.03,A -85,B 0,C 180,E1 12338.56,E2 12338.56} C_VEL
LIN {X 0,Y 506.456,Z 923.03,A -85,B 0,C 180,E1 12343.793,E2 12343.793} C_VEL
LIN {X 0,Y 506.251,Z 923.03,A -85,B 0,C 180,E1 12349.15,E2 12349.15} C_VEL
LIN {X 0,Y 506.002,Z 923.03,A -85,B 0,C 180,E1 12354.695,E2 12354.695} C_VEL
LIN {X 0,Y 505.915,Z 923.03,A -85,B 0,C 180,E1 12360.494,E2 12360.494} C_VEL
LIN {X 0,Y 505.742,Z 923.03,A -85,B 0,C 180,E1 12366.674,E2 12366.674} C_VEL
LIN {X 0,Y 505.679,Z 923.03,A -85,B 0,C 180,E1 12373.391,E2 12373.391} C_VEL
LIN {X 0,Y 505.64,Z 923.03,A -85,B 0,C 180,E1 12378.891,E2 12378.891} C_VEL
LIN {X 0,Y 505.752,Z 923.03,A -85,B 0,C 180,E1 12385.409,E2 12385.409} C_VEL
LIN {X 0,Y 505.791,Z 923.03,A -85,B 0,C 180,E1 12386.206,E2 12386.206} C_VEL
